LIN {X 0,Y 162.118,Z 704.88,A -85,B 0,C 180,E1 -25521.787,E2 -25521.787} C_VEL
LIN {X 0,Y 165.907,Z 693.035,A -85,B 0,C 180,E1 -25523.34,E2 -25523.34} C_VEL
LIN {X 0,Y 169.008,Z 680.232,A -85,B 0,C 180,E1 -25524.51,E2 -25524.51} C_VEL
LIN {X 0,Y 171.187,Z 667.318,A -85,B 0,C 180,E1 -25525.271,E2 -25525.271} C_VEL
LIN {X 0,Y 173.639,Z 638.606,A -85,B 0,C 180,E1 -25526.285,E2 -25526.285} C_VEL
LIN {X 0,Y 171.957,Z 634.293,A -85,B 0,C 180,E1 -25527.385,E2 -25527.385} C_VEL
LIN {X 0,Y 167.291,Z 625.497,A -85,B 0,C 180,E1 -25530.485,E2 -25530.485} C_VEL
LIN {X 0,Y 162.834,Z 618.085,A -85,B 0,C 180,E1 -25533.829,E2 -25533.829} C_VEL
LIN {X 0,Y 158.773,Z 611.768,A -85,B 0,C 180,E1 -25537.384,E2 -25537.384} C_VEL
LIN {X 0,Y 156.111,Z 607.869,A -85,B 0,C 180,E1 -25540.095,E2 -25540.095} C_VEL
LIN {X 0,Y 153.27,Z 603.781,A -85,B 0,C 180,E1 -25543.517,E2 -25543.517} C_VEL
LIN {X 0,Y 150.908,Z 600.619,A -85,B 0,C 180,E1 -25547.017,E2 -25547.017} C_VEL
LIN {X 0,Y 150.151,Z 599.126,A -85,B 0,C 180,E1 -25548.448,E2 -25548.448} C_VEL
LIN {X 0,Y 147.441,Z 595.958,A -85,B 0,C 180,E1 -25555.215,E2 -25555.215} C_VEL
LIN {X 0,Y 146.954,Z 593.781,A -85,B 0,C 180,E1 -25558.629,E2 -25558.629} C_VEL
LIN {X 0,Y 146.959,Z 593.9,A -85,B 0,C 180,E1 -25565.144,E2 -25565.144} C_VEL
LIN {X 0,Y 148.425,Z 597.823,A -85,B 0,C 180,E1 -25571.678,E2 -25571.678} C_VEL
LIN {X 0,Y 150.347,Z 599.549,A -85,B 0,C 180,E1 -25575.592,E2 -25575.592} C_VEL
LIN {X 0,Y 152.295,Z 602.878,A -85,B 0,C 180,E1 -25578.846,E2 -25578.846} C_VEL
LIN {X 0,Y 153.871,Z 604.601,A -85,B 0,C 180,E1 -25580.906,E2 -25580.906} C_VEL
LIN {X 0,Y 156.542,Z 608.421,A -85,B 0,C 180,E1 -25584.008,E2 -25584.008} C_VEL
LIN {X 0,Y 159.371,Z 612.825,A -85,B 0,C 180,E1 -25586.839,E2 -25586.839} C_VEL
LIN {X 0,Y 163.358,Z 620.37,A -85,B 0,C 180,E1 -25590.365,E2 -25590.365} C_VEL
LIN {X 0,Y 168.135,Z 630.963,A -85,B 0,C 180,E1 -25594.059,E2 -25594.059} C_VEL
LIN {X 0,Y 172.255,Z 641.448,A -85,B 0,C 180,E1 -25596.915,E2 -25596.915} C_VEL
LIN {X 0,Y 173.197,Z 644.283,A -85,B 0,C 180,E1 -25597.553,E2 -25597.553} C_VEL
LIN {X 0,Y 170.754,Z 672.948,A -85,B 0,C 180,E1 -25598.556,E2 -25598.556} C_VEL
LIN {X 0,Y 168.387,Z 686.79,A -85,B 0,C 180,E1 -25599.366,E2 -25599.366} C_VEL
LIN {X 0,Y 165.189,Z 699.4,A -85,B 0,C 180,E1 -25600.494,E2 -25600.494} C_VEL
LIN {X 0,Y 160.856,Z 711.897,A -85,B 0,C 180,E1 -25602.035,E2 -25602.035} C_VEL
LIN {X 0,Y 156.12,Z 723.049,A -85,B 0,C 180,E1 -25603.925,E2 -25603.925} C_VEL
LIN {X 0,Y 151.618,Z 732.079,A -85,B 0,C 180,E1 -25605.95,E2 -25605.95} C_VEL
LIN {X 0,Y 146.276,Z 741.359,A -85,B 0,C 180,E1 -25608.653,E2 -25608.653} C_VEL
LIN {X 0,Y 140.348,Z 750.363,A -85,B 0,C 180,E1 -25612.164,E2 -25612.164} C_VEL
LIN {X 0,Y 135.119,Z 757.631,A -85,B 0,C 180,E1 -25616.005,E2 -25616.005} C_VEL
LIN {X 0,Y 129.943,Z 764.292,A -85,B 0,C 180,E1 -25620.872,E2 -25620.872} C_VEL
LIN {X 0,Y 126.155,Z 768.706,A -85,B 0,C 180,E1 -25625.304,E2 -25625.304} C_VEL
LIN {X 0,Y 123.114,Z 772.057,A -85,B 0,C 180,E1 -25629.971,E2 -25629.971} C_VEL
LIN {X 0,Y 120.562,Z 775.013,A -85,B 0,C 180,E1 -25636.516,E2 -25636.516} C_VEL
LIN {X 0,Y 119.8,Z 775.898,A -85,B 0,C 180,E1 -25639.864,E2 -25639.864} C_VEL
LIN {X 0,Y 119.372,Z 776.351,A -85,B 0,C 180,E1 -25643.238,E2 -25643.238} C_VEL
LIN {X 0,Y 119.224,Z 776.413,A -85,B 0,C 180,E1 -25646.621,E2 -25646.621} C_VEL
LIN {X 0,Y 119.36,Z 776.091,A -85,B 0,C 180,E1 -25650,E2 -25650} C_VEL
LIN {X 0,Y 119.284,Z 775.366,A -85,B 0,C 180,E1 -25653.378,E2 -25653.378} C_VEL
LIN {X 0,Y 119.406,Z 774.199,A -85,B 0,C 180,E1 -25656.76,E2 -25656.76} C_VEL
LIN {X 0,Y 120.072,Z 771.674,A -85,B 0,C 180,E1 -25661.821,E2 -25661.821} C_VEL
LIN {X 0,Y 121.494,Z 768.132,A -85,B 0,C 180,E1 -25666.812,E2 -25666.812} C_VEL
LIN {X 0,Y 123.837,Z 763.485,A -85,B 0,C 180,E1 -25671.647,E2 -25671.647} C_VEL
LIN {X 0,Y 127.337,Z 756.895,A -85,B 0,C 180,E1 -25676.744,E2 -25676.744} C_VEL
LIN {X 0,Y 128.513,Z 753.671,A -85,B 0,C 180,E1 -25678.89,E2 -25678.89} C_VEL
LIN {X 0,Y 128.84,Z 748.046,A -85,B 0,C 180,E1 -25682.527,E2 -25682.527} C_VEL
LIN {X 0,Y 129.411,Z 741.896,A -85,B 0,C 180,E1 -25685.979,E2 -25685.979} C_VEL
LIN {X 0,Y 130.899,Z 737.763,A -85,B 0,C 180,E1 -25687.745,E2 -25687.745} C_VEL
LIN {X 0,Y 135.517,Z 727.836,A -85,B 0,C 180,E1 -25690.899,E2 -25690.899} C_VEL
LIN {X 0,Y 140.137,Z 716.363,A -85,B 0,C 180,E1 -25693.595,E2 -25693.595} C_VEL
LIN {X 0,Y 143.954,Z 705.097,A -85,B 0,C 180,E1 -25695.561,E2 -25695.561} C_VEL
LIN {X 0,Y 147.364,Z 692.405,A -85,B 0,C 180,E1 -25697.159,E2 -25697.159} C_VEL
LIN {X 0,Y 149.806,Z 679.678,A -85,B 0,C 180,E1 -25698.263,E2 -25698.263} C_VEL
LIN {X 0,Y 151.379,Z 666.349,A -85,B 0,C 180,E1 -25698.991,E2 -25698.991} C_VEL
LIN {X 0,Y 153.858,Z 633.14,A -85,B 0,C 180,E1 -25700.246,E2 -25700.246} C_VEL
LIN {X 0,Y 150.172,Z 622.407,A -85,B 0,C 180,E1 -25702.622,E2 -25702.622} C_VEL
LIN {X 0,Y 145.722,Z 611.956,A -85,B 0,C 180,E1 -25705.632,E2 -25705.632} C_VEL
LIN {X 0,Y 142.708,Z 605.888,A -85,B 0,C 180,E1 -25707.827,E2 -25707.827} C_VEL
LIN {X 0,Y 138.817,Z 599.957,A -85,B 0,C 180,E1 -25710.828,E2 -25710.828} C_VEL
LIN {X 0,Y 136.129,Z 596.114,A -85,B 0,C 180,E1 -25713.145,E2 -25713.145} C_VEL
LIN {X 0,Y 133.127,Z 591.974,A -85,B 0,C 180,E1 -25716.057,E2 -25716.057} C_VEL
LIN {X 0,Y 130.457,Z 588.575,A -85,B 0,C 180,E1 -25719.022,E2 -25719.022} C_VEL
LIN {X 0,Y 129.642,Z 587.229,A -85,B 0,C 180,E1 -25720.072,E2 -25720.072} C_VEL
LIN {X 0,Y 127.258,Z 584.922,A -85,B 0,C 180,E1 -25723.275,E2 -25723.275} C_VEL
LIN {X 0,Y 125.817,Z 582.049,A -85,B 0,C 180,E1 -25725.855,E2 -25725.855} C_VEL
LIN {X 0,Y 122.518,Z 579.199,A -85,B 0,C 180,E1 -25733.413,E2 -25733.413} C_VEL
LIN {X 0,Y 121.752,Z 576.723,A -85,B 0,C 180,E1 -25737.726,E2 -25737.726} C_VEL
LIN {X 0,Y 121.716,Z 576.23,A -85,B 0,C 180,E1 -25738.346,E2 -25738.346} C_VEL
LIN {X 0,Y 121.562,Z 576.369,A -85,B 0,C 180,E1 -25744.975,E2 -25744.975} C_VEL
LIN {X 0,Y 123.992,Z 581.142,A -85,B 0,C 180,E1 -25755.198,E2 -25755.198} C_VEL
LIN {X 0,Y 125.934,Z 582.245,A -85,B 0,C 180,E1 -25758.822,E2 -25758.822} C_VEL
LIN {X 0,Y 127.529,Z 585.423,A -85,B 0,C 180,E1 -25761.618,E2 -25761.618} C_VEL
LIN {X 0,Y 130.086,Z 587.796,A -85,B 0,C 180,E1 -25764.94,E2 -25764.94} C_VEL
LIN {X 0,Y 132.291,Z 591.204,A -85,B 0,C 180,E1 -25767.556,E2 -25767.556} C_VEL
LIN {X 0,Y 133.801,Z 592.774,A -85,B 0,C 180,E1 -25769.076,E2 -25769.076} C_VEL
LIN {X 0,Y 136.478,Z 596.545,A -85,B 0,C 180,E1 -25771.621,E2 -25771.621} C_VEL
LIN {X 0,Y 140.346,Z 602.297,A -85,B 0,C 180,E1 -25774.859,E2 -25774.859} C_VEL
LIN {X 0,Y 144.7,Z 609.144,A -85,B 0,C 180,E1 -25778.042,E2 -25778.042} C_VEL
LIN {X 0,Y 149.212,Z 617.122,A -85,B 0,C 180,E1 -25780.99,E2 -25780.99} C_VEL
LIN {X 0,Y 153.985,Z 626.915,A -85,B 0,C 180,E1 -25783.837,E2 -25783.837} C_VEL
LIN {X 0,Y 154.23,Z 628.253,A -85,B 0,C 180,E1 -25784.032,E2 -25784.032} C_VEL
LIN {X 0,Y 151.162,Z 666.895,A -85,B 0,C 180,E1 -25785.536,E2 -25785.536} C_VEL
LIN {X 0,Y 149.109,Z 680.278,A -85,B 0,C 180,E1 -25786.482,E2 -25786.482} C_VEL
LIN {X 0,Y 146.492,Z 692.384,A -85,B 0,C 180,E1 -25787.807,E2 -25787.807} C_VEL
LIN {X 0,Y 143.233,Z 703.52,A -85,B 0,C 180,E1 -25789.449,E2 -25789.449} C_VEL
LIN {X 0,Y 139.286,Z 715.044,A -85,B 0,C 180,E1 -25791.823,E2 -25791.823} C_VEL
LIN {X 0,Y 134.978,Z 725.424,A -85,B 0,C 180,E1 -25794.603,E2 -25794.603} C_VEL
LIN {X 0,Y 130.826,Z 733.925,A -85,B 0,C 180,E1 -25797.507,E2 -25797.507} C_VEL
LIN {X 0,Y 126.685,Z 741.757,A -85,B 0,C 180,E1 -25800.961,E2 -25800.961} C_VEL
LIN {X 0,Y 122.587,Z 749.395,A -85,B 0,C 180,E1 -25805.441,E2 -25805.441} C_VEL
LIN {X 0,Y 118.556,Z 756.43,A -85,B 0,C 180,E1 -25810.972,E2 -25810.972} C_VEL
LIN {X 0,Y 115.874,Z 761.117,A -85,B 0,C 180,E1 -25815.96,E2 -25815.96} C_VEL
LIN {X 0,Y 113.867,Z 764.711,A -85,B 0,C 180,E1 -25821.124,E2 -25821.124} C_VEL
LIN {X 0,Y 112.581,Z 767.627,A -85,B 0,C 180,E1 -25827.226,E2 -25827.226} C_VEL
LIN {X 0,Y 112.176,Z 769.339,A -85,B 0,C 180,E1 -25833.592,E2 -25833.592} C_VEL
LIN {X 0,Y 112.24,Z 769.739,A -85,B 0,C 180,E1 -25837.194,E2 -25837.194} C_VEL
LIN {X 0,Y 112.619,Z 769.76,A -85,B 0,C 180,E1 -25840.79,E2 -25840.79} C_VEL
LIN {X 0,Y 113.276,Z 769.401,A -85,B 0,C 180,E1 -25844.369,E2 -25844.369} C_VEL
LIN {X 0,Y 114.271,Z 768.638,A -85,B 0,C 180,E1 -25847.909,E2 -25847.909} C_VEL
LIN {X 0,Y 117.478,Z 765.84,A -85,B 0,C 180,E1 -25854.756,E2 -25854.756} C_VEL
LIN {X 0,Y 120.696,Z 762.736,A -85,B 0,C 180,E1 -25859.474,E2 -25859.474} C_VEL
LIN {X 0,Y 124.879,Z 758.31,A -85,B 0,C 180,E1 -25864.248,E2 -25864.248} C_VEL
LIN {X 0,Y 129.683,Z 752.804,A -85,B 0,C 180,E1 -25868.551,E2 -25868.551} C_VEL
LIN {X 0,Y 135.205,Z 745.915,A -85,B 0,C 180,E1 -25872.511,E2 -25872.511} C_VEL
LIN {X 0,Y 140.125,Z 738.86,A -85,B 0,C 180,E1 -25875.618,E2 -25875.618} C_VEL
LIN {X 0,Y 145.46,Z 730.317,A -85,B 0,C 180,E1 -25878.493,E2 -25878.493} C_VEL
LIN {X 0,Y 150.579,Z 720.926,A -85,B 0,C 180,E1 -25880.889,E2 -25880.889} C_VEL
LIN {X 0,Y 155.981,Z 709.252,A -85,B 0,C 180,E1 -25883.105,E2 -25883.105} C_VEL
LIN {X 0,Y 160.204,Z 697.641,A -85,B 0,C 180,E1 -25884.79,E2 -25884.79} C_VEL
LIN {X 0,Y 163.634,Z 685.457,A -85,B 0,C 180,E1 -25886.058,E2 -25886.058} C_VEL
LIN {X 0,Y 166.304,Z 672.324,A -85,B 0,C 180,E1 -25886.991,E2 -25886.991} C_VEL
LIN {X 0,Y 167.9,Z 659.529,A -85,B 0,C 180,E1 -25887.531,E2 -25887.531} C_VEL
LIN {X 0,Y 169.328,Z 640.85,A -85,B 0,C 180,E1 -25888.206,E2 -25888.206} C_VEL
LIN {X 0,Y 165.427,Z 632.926,A -85,B 0,C 180,E1 -25890.938,E2 -25890.938} C_VEL
LIN {X 0,Y 161.192,Z 625.29,A -85,B 0,C 180,E1 -25894.259,E2 -25894.259} C_VEL
LIN {X 0,Y 157.108,Z 618.499,A -85,B 0,C 180,E1 -25897.997,E2 -25897.997} C_VEL
LIN {X 0,Y 154.077,Z 614.001,A -85,B 0,C 180,E1 -25901.262,E2 -25901.262} C_VEL
LIN {X 0,Y 151.71,Z 610.394,A -85,B 0,C 180,E1 -25904.337,E2 -25904.337} C_VEL
LIN {X 0,Y 149.37,Z 606.945,A -85,B 0,C 180,E1 -25908.12,E2 -25908.12} C_VEL
LIN {X 0,Y 148.887,Z 605.947,A -85,B 0,C 180,E1 -25909.116,E2 -25909.116} C_VEL
LIN {X 0,Y 146.412,Z 602.783,A -85,B 0,C 180,E1 -25915.871,E2 -25915.871} C_VEL
LIN {X 0,Y 146.008,Z 600.763,A -85,B 0,C 180,E1 -25919.31,E2 -25919.31} C_VEL
LIN {X 0,Y 146.037,Z 601.034,A -85,B 0,C 180,E1 -25924.831,E2 -25924.831} C_VEL
LIN {X 0,Y 147.563,Z 604.989,A -85,B 0,C 180,E1 -25931.747,E2 -25931.747} C_VEL
LIN {X 0,Y 149.034,Z 606.321,A -85,B 0,C 180,E1 -25934.857,E2 -25934.857} C_VEL
LIN {X 0,Y 151.098,Z 609.827,A -85,B 0,C 180,E1 -25938.467,E2 -25938.467} C_VEL
LIN {X 0,Y 152.264,Z 611.208,A -85,B 0,C 180,E1 -25940.077,E2 -25940.077} C_VEL
LIN {X 0,Y 155.367,Z 615.93,A -85,B 0,C 180,E1 -25943.846,E2 -25943.846} C_VEL
LIN {X 0,Y 157.331,Z 619.197,A -85,B 0,C 180,E1 -25945.908,E2 -25945.908} C_VEL
LIN {X 0,Y 160.981,Z 626.578,A -85,B 0,C 180,E1 -25949.365,E2 -25949.365} C_VEL
LIN {X 0,Y 165.062,Z 636.16,A -85,B 0,C 180,E1 -25952.764,E2 -25952.764} C_VEL
LIN {X 0,Y 168.692,Z 645.914,A -85,B 0,C 180,E1 -25955.497,E2 -25955.497} C_VEL
LIN {X 0,Y 168.933,Z 646.687,A -85,B 0,C 180,E1 -25955.676,E2 -25955.676} C_VEL
LIN {X 0,Y 166.573,Z 673.039,A -85,B 0,C 180,E1 -25956.609,E2 -25956.609} C_VEL
LIN {X 0,Y 164.128,Z 686.751,A -85,B 0,C 180,E1 -25957.406,E2 -25957.406} C_VEL
LIN {X 0,Y 161.016,Z 698.742,A -85,B 0,C 180,E1 -25958.472,E2 -25958.472} C_VEL
LIN {X 0,Y 156.829,Z 710.545,A -85,B 0,C 180,E1 -25959.878,E2 -25959.878} C_VEL
LIN {X 0,Y 152.527,Z 720.615,A -85,B 0,C 180,E1 -25961.519,E2 -25961.519} C_VEL
LIN {X 0,Y 147.209,Z 731.097,A -85,B 0,C 180,E1 -25963.774,E2 -25963.774} C_VEL
LIN {X 0,Y 142.094,Z 739.672,A -85,B 0,C 180,E1 -25966.178,E2 -25966.178} C_VEL
LIN {X 0,Y 136.811,Z 747.585,A -85,B 0,C 180,E1 -25969.084,E2 -25969.084} C_VEL
LIN {X 0,Y 131.026,Z 755.339,A -85,B 0,C 180,E1 -25972.885,E2 -25972.885} C_VEL
LIN {X 0,Y 125.275,Z 762.475,A -85,B 0,C 180,E1 -25977.796,E2 -25977.796} C_VEL
LIN {X 0,Y 120.945,Z 767.245,A -85,B 0,C 180,E1 -25982.299,E2 -25982.299} C_VEL
LIN {X 0,Y 117.455,Z 770.911,A -85,B 0,C 180,E1 -25987.113,E2 -25987.113} C_VEL
LIN {X 0,Y 114.859,Z 773.578,A -85,B 0,C 180,E1 -25992.186,E2 -25992.186} C_VEL
LIN {X 0,Y 113.653,Z 774.846,A -85,B 0,C 180,E1 -25995.68,E2 -25995.68} C_VEL
LIN {X 0,Y 112.791,Z 775.714,A -85,B 0,C 180,E1 -25999.227,E2 -25999.227} C_VEL
LIN {X 0,Y 112.3,Z 776.151,A -85,B 0,C 180,E1 -26002.81,E2 -26002.81} C_VEL
LIN {X 0,Y 112.132,Z 776.202,A -85,B 0,C 180,E1 -26006.407,E2 -26006.407} C_VEL
LIN {X 0,Y 112.261,Z 775.87,A -85,B 0,C 180,E1 -26010,E2 -26010} C_VEL
LIN {X 0,Y 112.181,Z 775.131,A -85,B 0,C 180,E1 -26013.592,E2 -26013.592} C_VEL
LIN {X 0,Y 112.325,Z 773.944,A -85,B 0,C 180,E1 -26017.188,E2 -26017.188} C_VEL
LIN {X 0,Y 113.119,Z 771.397,A -85,B 0,C 180,E1 -26022.559,E2 -26022.559} C_VEL
LIN {X 0,Y 114.666,Z 767.829,A -85,B 0,C 180,E1 -26027.845,E2 -26027.845} C_VEL
LIN {X 0,Y 117.227,Z 763.156,A -85,B 0,C 180,E1 -26032.934,E2 -26032.934} C_VEL
LIN {X 0,Y 121.3,Z 756.107,A -85,B 0,C 180,E1 -26038.554,E2 -26038.554} C_VEL
LIN {X 0,Y 125.585,Z 748.276,A -85,B 0,C 180,E1 -26043.195,E2 -26043.195} C_VEL
LIN {X 0,Y 130.351,Z 738.851,A -85,B 0,C 180,E1 -26047.34,E2 -26047.34} C_VEL
LIN {X 0,Y 130.899,Z 737.763,A -85,B 0,C 180,E1 -26047.745,E2 -26047.745} C_VEL
LIN {X 0,Y 132.468,Z 733.502,A -85,B 0,C 180,E1 -26049.393,E2 -26049.393} C_VEL
LIN {X 0,Y 133.545,Z 726.254,A -85,B 0,C 180,E1 -26052.276,E2 -26052.276} C_VEL
LIN {X 0,Y 134.543,Z 718.538,A -85,B 0,C 180,E1 -26054.911,E2 -26054.911} C_VEL
LIN {X 0,Y 135.908,Z 713.543,A -85,B 0,C 180,E1 -26056.123,E2 -26056.123} C_VEL
LIN {X 0,Y 139.62,Z 702.498,A -85,B 0,C 180,E1 -26057.94,E2 -26057.94} C_VEL
LIN {X 0,Y 142.901,Z 690.176,A -85,B 0,C 180,E1 -26059.395,E2 -26059.395} C_VEL
LIN {X 0,Y 145.439,Z 676.771,A -85,B 0,C 180,E1 -26060.475,E2 -26060.475} C_VEL
LIN {X 0,Y 147.034,Z 661.516,A -85,B 0,C 180,E1 -26061.184,E2 -26061.184} C_VEL
LIN {X 0,Y 149.056,Z 635.163,A -85,B 0,C 180,E1 -26062.197,E2 -26062.197} C_VEL
LIN {X 0,Y 145.717,Z 625.389,A -85,B 0,C 180,E1 -26064.558,E2 -26064.558} C_VEL
LIN {X 0,Y 141.696,Z 615.626,A -85,B 0,C 180,E1 -26067.569,E2 -26067.569} C_VEL
LIN {X 0,Y 139.318,Z 610.734,A -85,B 0,C 180,E1 -26069.469,E2 -26069.469} C_VEL
LIN {X 0,Y 135.869,Z 605.405,A -85,B 0,C 180,E1 -26072.36,E2 -26072.36} C_VEL
LIN {X 0,Y 133.665,Z 602.102,A -85,B 0,C 180,E1 -26074.423,E2 -26074.423} C_VEL
LIN {X 0,Y 130.973,Z 598.258,A -85,B 0,C 180,E1 -26077.236,E2 -26077.236} C_VEL
LIN {X 0,Y 128.33,Z 594.498,A -85,B 0,C 180,E1 -26080.459,E2 -26080.459} C_VEL
LIN {X 0,Y 127.249,Z 593.323,A -85,B 0,C 180,E1 -26081.901,E2 -26081.901} C_VEL
LIN {X 0,Y 125.12,Z 590.482,A -85,B 0,C 180,E1 -26085.268,E2 -26085.268} C_VEL
LIN {X 0,Y 124.286,Z 588.847,A -85,B 0,C 180,E1 -26086.928,E2 -26086.928} C_VEL
LIN {X 0,Y 121.121,Z 585.317,A -85,B 0,C 180,E1 -26095.633,E2 -26095.633} C_VEL
LIN {X 0,Y 120.763,Z 583.221,A -85,B 0,C 180,E1 -26099.063,E2 -26099.063} C_VEL
LIN {X 0,Y 120.66,Z 583.415,A -85,B 0,C 180,E1 -26104.594,E2 -26104.594} C_VEL
LIN {X 0,Y 122.966,Z 588.141,A -85,B 0,C 180,E1 -26114.904,E2 -26114.904} C_VEL
LIN {X 0,Y 124.511,Z 589.209,A -85,B 0,C 180,E1 -26117.98,E2 -26117.98} C_VEL
LIN {X 0,Y 126.347,Z 592.521,A -85,B 0,C 180,E1 -26121.282,E2 -26121.282} C_VEL
LIN {X 0,Y 128.309,Z 594.45,A -85,B 0,C 180,E1 -26123.967,E2 -26123.967} C_VEL
LIN {X 0,Y 130.779,Z 598.091,A -85,B 0,C 180,E1 -26127.016,E2 -26127.016} C_VEL
LIN {X 0,Y 131.935,Z 599.597,A -85,B 0,C 180,E1 -26128.268,E2 -26128.268} C_VEL
LIN {X 0,Y 135.326,Z 604.562,A -85,B 0,C 180,E1 -26131.605,E2 -26131.605} C_VEL
LIN {X 0,Y 139.788,Z 611.578,A -85,B 0,C 180,E1 -26135.366,E2 -26135.366} C_VEL
LIN {X 0,Y 144.244,Z 619.402,A -85,B 0,C 180,E1 -26138.642,E2 -26138.642} C_VEL
LIN {X 0,Y 148.524,Z 628.114,A -85,B 0,C 180,E1 -26141.489,E2 -26141.489} C_VEL
LIN {X 0,Y 149.367,Z 629.964,A -85,B 0,C 180,E1 -26142.021,E2 -26142.021} C_VEL
LIN {X 0,Y 146.401,Z 666.845,A -85,B 0,C 180,E1 -26143.502,E2 -26143.502} C_VEL
LIN {X 0,Y 144.324,Z 680.033,A -85,B 0,C 180,E1 -26144.43,E2 -26144.43} C_VEL
LIN {X 0,Y 141.609,Z 692.171,A -85,B 0,C 180,E1 -26145.749,E2 -26145.749} C_VEL
LIN {X 0,Y 137.946,Z 704.19,A -85,B 0,C 180,E1 -26147.543,E2 -26147.543} C_VEL
LIN {X 0,Y 133.81,Z 715.628,A -85,B 0,C 180,E1 -26149.956,E2 -26149.956} C_VEL
LIN {X 0,Y 129.271,Z 725.945,A -85,B 0,C 180,E1 -26152.785,E2 -26152.785} C_VEL
LIN {X 0,Y 124.925,Z 734.392,A -85,B 0,C 180,E1 -26155.767,E2 -26155.767} C_VEL
LIN {X 0,Y 120.559,Z 742.177,A -85,B 0,C 180,E1 -26159.331,E2 -26159.331} C_VEL
LIN {X 0,Y 116.199,Z 749.764,A -85,B 0,C 180,E1 -26163.993,E2 -26163.993} C_VEL
LIN {X 0,Y 111.886,Z 756.768,A -85,B 0,C 180,E1 -26169.79,E2 -26169.79} C_VEL
LIN {X 0,Y 109.024,Z 761.427,A -85,B 0,C 180,E1 -26175.058,E2 -26175.058} C_VEL
LIN {X 0,Y 106.875,Z 764.995,A -85,B 0,C 180,E1 -26180.538,E2 -26180.538} C_VEL
LIN {X 0,Y 105.625,Z 767.56,A -85,B 0,C 180,E1 -26186.185,E2 -26186.185} C_VEL
LIN {X 0,Y 105.222,Z 768.772,A -85,B 0,C 180,E1 -26190,E2 -26190} C_VEL
LIN {X 0,Y 105.09,Z 769.561,A -85,B 0,C 180,E1 -26193.834,E2 -26193.834} C_VEL
LIN {X 0,Y 105.607,Z 769.96,A -85,B 0,C 180,E1 -26201.516,E2 -26201.516} C_VEL
LIN {X 0,Y 106.366,Z 769.589,A -85,B 0,C 180,E1 -26205.325,E2 -26205.325} C_VEL
LIN {X 0,Y 107.48,Z 768.803,A -85,B 0,C 180,E1 -26209.083,E2 -26209.083} C_VEL
LIN {X 0,Y 111.021,Z 765.979,A -85,B 0,C 180,E1 -26216.303,E2 -26216.303} C_VEL
LIN {X 0,Y 114.641,Z 762.727,A -85,B 0,C 180,E1 -26221.404,E2 -26221.404} C_VEL
LIN {X 0,Y 119.028,Z 758.396,A -85,B 0,C 180,E1 -26226.188,E2 -26226.188} C_VEL
LIN {X 0,Y 124.187,Z 752.86,A -85,B 0,C 180,E1 -26230.602,E2 -26230.602} C_VEL
LIN {X 0,Y 130.021,Z 745.932,A -85,B 0,C 180,E1 -26234.642,E2 -26234.642} C_VEL
LIN {X 0,Y 135.216,Z 738.839,A -85,B 0,C 180,E1 -26237.786,E2 -26237.786} C_VEL
LIN {X 0,Y 140.822,Z 730.233,A -85,B 0,C 180,E1 -26240.673,E2 -26240.673} C_VEL
LIN {X 0,Y 146.19,Z 720.782,A -85,B 0,C 180,E1 -26243.056,E2 -26243.056} C_VEL
LIN {X 0,Y 151.803,Z 709.033,A -85,B 0,C 180,E1 -26245.26,E2 -26245.26} C_VEL
LIN {X 0,Y 156.202,Z 697.255,A -85,B 0,C 180,E1 -26246.927,E2 -26246.927} C_VEL
LIN {X 0,Y 160.011,Z 683.903,A -85,B 0,C 180,E1 -26248.261,E2 -26248.261} C_VEL
LIN {X 0,Y 162.54,Z 671.326,A -85,B 0,C 180,E1 -26249.105,E2 -26249.105} C_VEL
LIN {X 0,Y 164.297,Z 656.044,A -85,B 0,C 180,E1 -26249.693,E2 -26249.693} C_VEL
LIN {X 0,Y 165.281,Z 644.004,A -85,B 0,C 180,E1 -26250.116,E2 -26250.116} C_VEL
LIN {X 0,Y 161.383,Z 636.036,A -85,B 0,C 180,E1 -26253.139,E2 -26253.139} C_VEL
LIN {X 0,Y 157.306,Z 628.511,A -85,B 0,C 180,E1 -26256.758,E2 -26256.758} C_VEL
LIN {X 0,Y 154.155,Z 623.384,A -85,B 0,C 180,E1 -26260.005,E2 -26260.005} C_VEL
LIN {X 0,Y 152.317,Z 620.42,A -85,B 0,C 180,E1 -26262.2,E2 -26262.2} C_VEL
LIN {X 0,Y 150.209,Z 617.008,A -85,B 0,C 180,E1 -26265.139,E2 -26265.139} C_VEL
LIN {X 0,Y 147.978,Z 613.477,A -85,B 0,C 180,E1 -26269.048,E2 -26269.048} C_VEL
LIN {X 0,Y 147.655,Z 612.811,A -85,B 0,C 180,E1 -26269.764,E2 -26269.764} C_VEL
LIN {X 0,Y 145.347,Z 609.414,A -85,B 0,C 180,E1 -26276.881,E2 -26276.881} C_VEL
LIN {X 0,Y 145.084,Z 607.736,A -85,B 0,C 180,E1 -26280,E2 -26280} C_VEL
LIN {X 0,Y 145.126,Z 608.106,A -85,B 0,C 180,E1 -26284.513,E2 -26284.513} C_VEL
LIN {X 0,Y 146.558,Z 611.977,A -85,B 0,C 180,E1 -26291.443,E2 -26291.443} C_VEL
LIN {X 0,Y 147.821,Z 613.259,A -85,B 0,C 180,E1 -26294.278,E2 -26294.278} C_VEL
LIN {X 0,Y 150.016,Z 616.928,A -85,B 0,C 180,E1 -26298.246,E2 -26298.246} C_VEL
LIN {X 0,Y 150.811,Z 618.052,A -85,B 0,C 180,E1 -26299.414,E2 -26299.414} C_VEL
LIN {X 0,Y 153.565,Z 622.404,A -85,B 0,C 180,E1 -26302.961,E2 -26302.961} C_VEL
LIN {X 0,Y 155.319,Z 625.553,A -85,B 0,C 180,E1 -26304.938,E2 -26304.938} C_VEL
LIN {X 0,Y 158.636,Z 632.734,A -85,B 0,C 180,E1 -26308.316,E2 -26308.316} C_VEL
LIN {X 0,Y 162.266,Z 641.896,A -85,B 0,C 180,E1 -26311.584,E2 -26311.584} C_VEL
LIN {X 0,Y 164.853,Z 649.208,A -85,B 0,C 180,E1 -26313.711,E2 -26313.711} C_VEL
LIN {X 0,Y 162.636,Z 672.86,A -85,B 0,C 180,E1 -26314.552,E2 -26314.552} C_VEL
LIN {X 0,Y 160.16,Z 686.381,A -85,B 0,C 180,E1 -26315.331,E2 -26315.331} C_VEL
LIN {X 0,Y 156.708,Z 699.085,A -85,B 0,C 180,E1 -26316.444,E2 -26316.444} C_VEL
LIN {X 0,Y 152.391,Z 710.773,A -85,B 0,C 180,E1 -26317.837,E2 -26317.837} C_VEL
LIN {X 0,Y 147.915,Z 720.765,A -85,B 0,C 180,E1 -26319.459,E2 -26319.459} C_VEL
LIN {X 0,Y 142.398,Z 731.185,A -85,B 0,C 180,E1 -26321.714,E2 -26321.714} C_VEL
LIN {X 0,Y 137.062,Z 739.711,A -85,B 0,C 180,E1 -26324.123,E2 -26324.123} C_VEL
LIN {X 0,Y 131.536,Z 747.584,A -85,B 0,C 180,E1 -26327.061,E2 -26327.061} C_VEL
LIN {X 0,Y 125.418,Z 755.287,A -85,B 0,C 180,E1 -26330.92,E2 -26330.92} C_VEL
LIN {X 0,Y 120.084,Z 761.494,A -85,B 0,C 180,E1 -26335.218,E2 -26335.218} C_VEL
LIN {X 0,Y 114.679,Z 767.136,A -85,B 0,C 180,E1 -26340.642,E2 -26340.642} C_VEL
LIN {X 0,Y 110.936,Z 770.778,A -85,B 0,C 180,E1 -26345.683,E2 -26345.683} C_VEL
LIN {X 0,Y 108.077,Z 773.421,A -85,B 0,C 180,E1 -26351.027,E2 -26351.027} C_VEL
LIN {X 0,Y 106.761,Z 774.679,A -85,B 0,C 180,E1 -26354.733,E2 -26354.733} C_VEL
LIN {X 0,Y 105.812,Z 775.528,A -85,B 0,C 180,E1 -26358.507,E2 -26358.507} C_VEL
LIN {X 0,Y 105.252,Z 775.952,A -85,B 0,C 180,E1 -26362.326,E2 -26362.326} C_VEL
LIN {X 0,Y 105.04,Z 775.992,A -85,B 0,C 180,E1 -26366.164,E2 -26366.164} C_VEL
LIN {X 0,Y 105.173,Z 775.649,A -85,B 0,C 180,E1 -26370,E2 -26370} C_VEL
LIN {X 0,Y 105.097,Z 774.893,A -85,B 0,C 180,E1 -26373.834,E2 -26373.834} C_VEL
LIN {X 0,Y 105.267,Z 773.689,A -85,B 0,C 180,E1 -26377.673,E2 -26377.673} C_VEL
LIN {X 0,Y 106.157,Z 771.118,A -85,B 0,C 180,E1 -26383.398,E2 -26383.398} C_VEL
LIN {X 0,Y 107.884,Z 767.526,A -85,B 0,C 180,E1 -26389.009,E2 -26389.009} C_VEL
LIN {X 0,Y 110.692,Z 762.827,A -85,B 0,C 180,E1 -26394.374,E2 -26394.374} C_VEL
LIN {X 0,Y 114.369,Z 756.873,A -85,B 0,C 180,E1 -26399.445,E2 -26399.445} C_VEL
LIN {X 0,Y 118.746,Z 749.443,A -85,B 0,C 180,E1 -26404.209,E2 -26404.209} C_VEL
LIN {X 0,Y 123.816,Z 740.194,A -85,B 0,C 180,E1 -26408.636,E2 -26408.636} C_VEL
LIN {X 0,Y 129.181,Z 729.51,A -85,B 0,C 180,E1 -26412.317,E2 -26412.317} C_VEL
LIN {X 0,Y 133.951,Z 718.618,A -85,B 0,C 180,E1 -26415.096,E2 -26415.096} C_VEL
LIN {X 0,Y 135.908,Z 713.543,A -85,B 0,C 180,E1 -26416.123,E2 -26416.123} C_VEL
LIN {X 0,Y 137.179,Z 708.426,A -85,B 0,C 180,E1 -26417.262,E2 -26417.262} C_VEL
LIN {X 0,Y 137.771,Z 699.917,A -85,B 0,C 180,E1 -26419.439,E2 -26419.439} C_VEL
LIN {X 0,Y 138.237,Z 691.126,A -85,B 0,C 180,E1 -26421.318,E2 -26421.318} C_VEL
LIN {X 0,Y 139.21,Z 685.539,A -85,B 0,C 180,E1 -26421.962,E2 -26421.962} C_VEL
LIN {X 0,Y 141.398,Z 672.552,A -85,B 0,C 180,E1 -26422.862,E2 -26422.862} C_VEL
LIN {X 0,Y 144.429,Z 637.273,A -85,B 0,C 180,E1 -26424.273,E2 -26424.273} C_VEL
LIN {X 0,Y 141.408,Z 628.202,A -85,B 0,C 180,E1 -26426.646,E2 -26426.646} C_VEL
LIN {X 0,Y 137.488,Z 618.394,A -85,B 0,C 180,E1 -26429.934,E2 -26429.934} C_VEL
LIN {X 0,Y 134.313,Z 612.689,A -85,B 0,C 180,E1 -26432.753,E2 -26432.753} C_VEL
LIN {X 0,Y 130.882,Z 607.553,A -85,B 0,C 180,E1 -26436.159,E2 -26436.159} C_VEL
LIN {X 0,Y 128.932,Z 604.537,A -85,B 0,C 180,E1 -26438.399,E2 -26438.399} C_VEL
LIN {X 0,Y 126.105,Z 600.363,A -85,B 0,C 180,E1 -26442.177,E2 -26442.177} C_VEL
LIN {X 0,Y 123.74,Z 597.337,A -85,B 0,C 180,E1 -26446.045,E2 -26446.045} C_VEL
LIN {X 0,Y 122.977,Z 595.681,A -85,B 0,C 180,E1 -26447.695,E2 -26447.695} C_VEL
LIN {X 0,Y 120.102,Z 592.13,A -85,B 0,C 180,E1 -26456.41,E2 -26456.41} C_VEL
LIN {X 0,Y 119.813,Z 590.196,A -85,B 0,C 180,E1 -26460,E2 -26460} C_VEL
LIN {X 0,Y 119.757,Z 590.455,A -85,B 0,C 180,E1 -26464.122,E2 -26464.122} C_VEL
LIN {X 0,Y 121.867,Z 595.081,A -85,B 0,C 180,E1 -26474.424,E2 -26474.424} C_VEL
LIN {X 0,Y 123.174,Z 596.153,A -85,B 0,C 180,E1 -26477.217,E2 -26477.217} C_VEL
LIN {X 0,Y 124.999,Z 599.373,A -85,B 0,C 180,E1 -26480.664,E2 -26480.664} C_VEL
LIN {X 0,Y 126.612,Z 601.148,A -85,B 0,C 180,E1 -26483.025,E2 -26483.025} C_VEL
LIN {X 0,Y 129.255,Z 604.953,A -85,B 0,C 180,E1 -26486.436,E2 -26486.436} C_VEL
LIN {X 0,Y 132.812,Z 610.461,A -85,B 0,C 180,E1 -26490.285,E2 -26490.285} C_VEL
LIN {X 0,Y 136.777,Z 616.923,A -85,B 0,C 180,E1 -26493.904,E2 -26493.904} C_VEL
LIN {X 0,Y 140.997,Z 624.708,A -85,B 0,C 180,E1 -26497.273,E2 -26497.273} C_VEL
LIN {X 0,Y 144.711,Z 632.63,A -85,B 0,C 180,E1 -26499.959,E2 -26499.959} C_VEL
LIN {X 0,Y 141.737,Z 667.591,A -85,B 0,C 180,E1 -26501.382,E2 -26501.382} C_VEL
LIN {X 0,Y 139.588,Z 680.578,A -85,B 0,C 180,E1 -26502.312,E2 -26502.312} C_VEL
LIN {X 0,Y 136.634,Z 693.037,A -85,B 0,C 180,E1 -26503.683,E2 -26503.683} C_VEL
LIN {X 0,Y 132.82,Z 704.86,A -85,B 0,C 180,E1 -26505.485,E2 -26505.485} C_VEL
LIN {X 0,Y 128.472,Z 716.213,A -85,B 0,C 180,E1 -26507.924,E2 -26507.924} C_VEL
LIN {X 0,Y 123.711,Z 726.464,A -85,B 0,C 180,E1 -26510.802,E2 -26510.802} C_VEL
LIN {X 0,Y 119.153,Z 734.854,A -85,B 0,C 180,E1 -26513.856,E2 -26513.856} C_VEL
LIN {X 0,Y 113.71,Z 743.938,A -85,B 0,C 180,E1 -26518.309,E2 -26518.309} C_VEL
LIN {X 0,Y 109.166,Z 751.241,A -85,B 0,C 180,E1 -26523.215,E2 -26523.215} C_VEL
LIN {X 0,Y 105.266,Z 757.106,A -85,B 0,C 180,E1 -26528.457,E2 -26528.457} C_VEL
LIN {X 0,Y 102.192,Z 761.737,A -85,B 0,C 180,E1 -26534.033,E2 -26534.033} C_VEL
LIN {X 0,Y 99.895,Z 765.278,A -85,B 0,C 180,E1 -26539.87,E2 -26539.87} C_VEL
LIN {X 0,Y 98.562,Z 767.818,A -85,B 0,C 180,E1 -26545.911,E2 -26545.911} C_VEL
LIN {X 0,Y 98.14,Z 769.016,A -85,B 0,C 180,E1 -26550,E2 -26550} C_VEL
LIN {X 0,Y 98.001,Z 769.784,A -85,B 0,C 180,E1 -26554.112,E2 -26554.112} C_VEL
LIN {X 0,Y 98.628,Z 770.159,A -85,B 0,C 180,E1 -26562.343,E2 -26562.343} C_VEL
LIN {X 0,Y 99.498,Z 769.777,A -85,B 0,C 180,E1 -26566.411,E2 -26566.411} C_VEL
LIN {X 0,Y 100.74,Z 768.967,A -85,B 0,C 180,E1 -26570.414,E2 -26570.414} C_VEL
LIN {X 0,Y 102.515,Z 767.743,A -85,B 0,C 180,E1 -26574.288,E2 -26574.288} C_VEL
LIN {X 0,Y 106.851,Z 764.327,A -85,B 0,C 180,E1 -26581.232,E2 -26581.232} C_VEL
LIN {X 0,Y 111.662,Z 760.085,A -85,B 0,C 180,E1 -26586.721,E2 -26586.721} C_VEL
LIN {X 0,Y 117.858,Z 753.923,A -85,B 0,C 180,E1 -26592.132,E2 -26592.132} C_VEL
LIN {X 0,Y 123.971,Z 747.193,A -85,B 0,C 180,E1 -26596.285,E2 -26596.285} C_VEL
LIN {X 0,Y 130.504,Z 738.811,A -85,B 0,C 180,E1 -26600.119,E2 -26600.119} C_VEL
LIN {X 0,Y 136.404,Z 730.148,A -85,B 0,C 180,E1 -26602.996,E2 -26602.996} C_VEL
LIN {X 0,Y 142.027,Z 720.639,A -85,B 0,C 180,E1 -26605.351,E2 -26605.351} C_VEL
LIN {X 0,Y 147.204,Z 710.245,A -85,B 0,C 180,E1 -26607.294,E2 -26607.294} C_VEL
LIN {X 0,Y 151.762,Z 698.821,A -85,B 0,C 180,E1 -26608.949,E2 -26608.949} C_VEL
LIN {X 0,Y 155.504,Z 686.697,A -85,B 0,C 180,E1 -26610.208,E2 -26610.208} C_VEL
LIN {X 0,Y 158.524,Z 672.973,A -85,B 0,C 180,E1 -26611.174,E2 -26611.174} C_VEL
LIN {X 0,Y 160.277,Z 660.038,A -85,B 0,C 180,E1 -26611.702,E2 -26611.702} C_VEL
LIN {X 0,Y 161.344,Z 647.14,A -85,B 0,C 180,E1 -26612.172,E2 -26612.172} C_VEL
LIN {X 0,Y 157.564,Z 639.279,A -85,B 0,C 180,E1 -26615.456,E2 -26615.456} C_VEL
LIN {X 0,Y 154.003,Z 632.691,A -85,B 0,C 180,E1 -26619.025,E2 -26619.025} C_VEL
LIN {X 0,Y 150.805,Z 627.112,A -85,B 0,C 180,E1 -26622.891,E2 -26622.891} C_VEL
LIN {X 0,Y 148.512,Z 623.365,A -85,B 0,C 180,E1 -26626.313,E2 -26626.313} C_VEL
LIN {X 0,Y 146.442,Z 619.669,A -85,B 0,C 180,E1 -26630.423,E2 -26630.423} C_VEL
LIN {X 0,Y 144.294,Z 615.857,A -85,B 0,C 180,E1 -26638.255,E2 -26638.255} C_VEL
LIN {X 0,Y 144.219,Z 614.776,A -85,B 0,C 180,E1 -26640,E2 -26640} C_VEL
LIN {X 0,Y 144.216,Z 615.073,A -85,B 0,C 180,E1 -26644.017,E2 -26644.017} C_VEL
LIN {X 0,Y 145.557,Z 618.959,A -85,B 0,C 180,E1 -26651.135,E2 -26651.135} C_VEL
LIN {X 0,Y 146.564,Z 620.024,A -85,B 0,C 180,E1 -26653.54,E2 -26653.54} C_VEL
LIN {X 0,Y 148.701,Z 623.733,A -85,B 0,C 180,E1 -26657.657,E2 -26657.657} C_VEL
LIN {X 0,Y 151.911,Z 629.021,A -85,B 0,C 180,E1 -26662.187,E2 -26662.187} C_VEL
LIN {X 0,Y 153.531,Z 632.273,A -85,B 0,C 180,E1 -26664.149,E2 -26664.149} C_VEL
LIN {X 0,Y 156.664,Z 639.637,A -85,B 0,C 180,E1 -26667.556,E2 -26667.556} C_VEL
LIN {X 0,Y 160.083,Z 649.171,A -85,B 0,C 180,E1 -26670.857,E2 -26670.857} C_VEL
LIN {X 0,Y 160.975,Z 651.803,A -85,B 0,C 180,E1 -26671.654,E2 -26671.654} C_VEL
LIN {X 0,Y 158.77,Z 673.737,A -85,B 0,C 180,E1 -26672.45,E2 -26672.45} C_VEL
LIN {X 0,Y 156.364,Z 686.126,A -85,B 0,C 180,E1 -26673.147,E2 -26673.147} C_VEL
LIN {X 0,Y 152.967,Z 698.43,A -85,B 0,C 180,E1 -26674.21,E2 -26674.21} C_VEL
LIN {X 0,Y 148.159,Z 711.001,A -85,B 0,C 180,E1 -26675.677,E2 -26675.677} C_VEL
LIN {X 0,Y 142.88,Z 722.203,A -85,B 0,C 180,E1 -26677.52,E2 -26677.52} C_VEL
LIN {X 0,Y 137.112,Z 732.299,A -85,B 0,C 180,E1 -26679.75,E2 -26679.75} C_VEL
LIN {X 0,Y 131.039,Z 741.411,A -85,B 0,C 180,E1 -26682.487,E2 -26682.487} C_VEL
LIN {X 0,Y 124.199,Z 750.303,A -85,B 0,C 180,E1 -26686.118,E2 -26686.118} C_VEL
LIN {X 0,Y 117.986,Z 757.466,A -85,B 0,C 180,E1 -26690.184,E2 -26690.184} C_VEL
LIN {X 0,Y 111.772,Z 764.006,A -85,B 0,C 180,E1 -26695.536,E2 -26695.536} C_VEL
LIN {X 0,Y 107.108,Z 768.344,A -85,B 0,C 180,E1 -26700.521,E2 -26700.521} C_VEL
LIN {X 0,Y 103.304,Z 771.623,A -85,B 0,C 180,E1 -26705.909,E2 -26705.909} C_VEL
LIN {X 0,Y 99.887,Z 774.511,A -85,B 0,C 180,E1 -26713.654,E2 -26713.654} C_VEL
LIN {X 0,Y 98.832,Z 775.339,A -85,B 0,C 180,E1 -26717.683,E2 -26717.683} C_VEL
LIN {X 0,Y 98.205,Z 775.752,A -85,B 0,C 180,E1 -26721.771,E2 -26721.771} C_VEL
LIN {X 0,Y 97.946,Z 775.782,A -85,B 0,C 180,E1 -26725.885,E2 -26725.885} C_VEL
LIN {X 0,Y 98.076,Z 775.428,A -85,B 0,C 180,E1 -26730,E2 -26730} C_VEL
LIN {X 0,Y 98.011,Z 774.653,A -85,B 0,C 180,E1 -26734.112,E2 -26734.112} C_VEL
LIN {X 0,Y 98.213,Z 773.434,A -85,B 0,C 180,E1 -26738.228,E2 -26738.228} C_VEL
LIN {X 0,Y 99.22,Z 770.839,A -85,B 0,C 180,E1 -26744.354,E2 -26744.354} C_VEL
LIN {X 0,Y 101.159,Z 767.223,A -85,B 0,C 180,E1 -26750.326,E2 -26750.326} C_VEL
LIN {X 0,Y 104.237,Z 762.497,A -85,B 0,C 180,E1 -26755.992,E2 -26755.992} C_VEL
LIN {X 0,Y 108.239,Z 756.515,A -85,B 0,C 180,E1 -26761.294,E2 -26761.294} C_VEL
LIN {X 0,Y 112.747,Z 749.321,A -85,B 0,C 180,E1 -26766.089,E2 -26766.089} C_VEL
LIN {X 0,Y 117.365,Z 741.433,A -85,B 0,C 180,E1 -26770.069,E2 -26770.069} C_VEL
LIN {X 0,Y 122.408,Z 732.217,A -85,B 0,C 180,E1 -26773.548,E2 -26773.548} C_VEL
LIN {X 0,Y 127.352,Z 721.965,A -85,B 0,C 180,E1 -26776.41,E2 -26776.41} C_VEL
LIN {X 0,Y 131.959,Z 710.58,A -85,B 0,C 180,E1 -26778.787,E2 -26778.787} C_VEL
LIN {X 0,Y 135.911,Z 698.755,A -85,B 0,C 180,E1 -26780.57,E2 -26780.57} C_VEL
LIN {X 0,Y 139.075,Z 686.086,A -85,B 0,C 180,E1 -26781.927,E2 -26781.927} C_VEL
LIN {X 0,Y 139.21,Z 685.539,A -85,B 0,C 180,E1 -26781.962,E2 -26781.962} C_VEL
LIN {X 0,Y 140.064,Z 679.872,A -85,B 0,C 180,E1 -26782.527,E2 -26782.527} C_VEL
LIN {X 0,Y 139.608,Z 670.64,A -85,B 0,C 180,E1 -26783.999,E2 -26783.999} C_VEL
LIN {X 0,Y 138.599,Z 661.317,A -85,B 0,C 180,E1 -26785.411,E2 -26785.411} C_VEL
LIN {X 0,Y 138.645,Z 655.487,A -85,B 0,C 180,E1 -26785.869,E2 -26785.869} C_VEL
LIN {X 0,Y 139.99,Z 639.533,A -85,B 0,C 180,E1 -26786.479,E2 -26786.479} C_VEL
LIN {X 0,Y 137.473,Z 631.638,A -85,B 0,C 180,E1 -26788.694,E2 -26788.694} C_VEL
LIN {X 0,Y 134.002,Z 622.581,A -85,B 0,C 180,E1 -26791.941,E2 -26791.941} C_VEL
LIN {X 0,Y 130.811,Z 617.07,A -85,B 0,C 180,E1 -26795.076,E2 -26795.076} C_VEL
LIN {X 0,Y 127.177,Z 611.134,A -85,B 0,C 180,E1 -26799.305,E2 -26799.305} C_VEL
LIN {X 0,Y 124.213,Z 606.708,A -85,B 0,C 180,E1 -26803.567,E2 -26803.567} C_VEL
LIN {X 0,Y 122.046,Z 603.427,A -85,B 0,C 180,E1 -26807.599,E2 -26807.599} C_VEL
LIN {X 0,Y 121.644,Z 602.498,A -85,B 0,C 180,E1 -26808.57,E2 -26808.57} C_VEL
LIN {X 0,Y 119.096,Z 598.937,A -85,B 0,C 180,E1 -26817.252,E2 -26817.252} C_VEL
LIN {X 0,Y 118.928,Z 597.396,A -85,B 0,C 180,E1 -26820,E2 -26820} C_VEL
LIN {X 0,Y 118.868,Z 597.474,A -85,B 0,C 180,E1 -26823.682,E2 -26823.682} C_VEL
LIN {X 0,Y 120.807,Z 602.017,A -85,B 0,C 180,E1 -26834.004,E2 -26834.004} C_VEL
LIN {X 0,Y 121.819,Z 602.976,A -85,B 0,C 180,E1 -26836.335,E2 -26836.335} C_VEL
LIN {X 0,Y 123.746,Z 606.301,A -85,B 0,C 180,E1 -26840.163,E2 -26840.163} C_VEL
LIN {X 0,Y 124.939,Z 607.788,A -85,B 0,C 180,E1 -26842.034,E2 -26842.034} C_VEL
LIN {X 0,Y 127.975,Z 612.506,A -85,B 0,C 180,E1 -26846.172,E2 -26846.172} C_VEL
LIN {X 0,Y 131.145,Z 617.576,A -85,B 0,C 180,E1 -26849.723,E2 -26849.723} C_VEL
LIN {X 0,Y 135.396,Z 625.215,A -85,B 0,C 180,E1 -26853.777,E2 -26853.777} C_VEL
LIN {X 0,Y 138.864,Z 632.315,A -85,B 0,C 180,E1 -26856.683,E2 -26856.683} C_VEL
LIN {X 0,Y 140.252,Z 635.337,A -85,B 0,C 180,E1 -26857.766,E2 -26857.766} C_VEL
LIN {X 0,Y 137.404,Z 667.437,A -85,B 0,C 180,E1 -26859.069,E2 -26859.069} C_VEL
LIN {X 0,Y 135.194,Z 680.44,A -85,B 0,C 180,E1 -26859.988,E2 -26859.988} C_VEL
LIN {X 0,Y 132.144,Z 692.87,A -85,B 0,C 180,E1 -26861.336,E2 -26861.336} C_VEL
LIN {X 0,Y 128.472,Z 703.956,A -85,B 0,C 180,E1 -26862.974,E2 -26862.974} C_VEL
LIN {X 0,Y 123.896,Z 715.513,A -85,B 0,C 180,E1 -26865.416,E2 -26865.416} C_VEL
LIN {X 0,Y 118.866,Z 725.92,A -85,B 0,C 180,E1 -26868.307,E2 -26868.307} C_VEL
LIN {X 0,Y 113.528,Z 735.308,A -85,B 0,C 180,E1 -26871.754,E2 -26871.754} C_VEL
LIN {X 0,Y 107.752,Z 744.341,A -85,B 0,C 180,E1 -26876.331,E2 -26876.331} C_VEL
LIN {X 0,Y 102.895,Z 751.61,A -85,B 0,C 180,E1 -26881.438,E2 -26881.438} C_VEL
LIN {X 0,Y 98.708,Z 757.444,A -85,B 0,C 180,E1 -26886.946,E2 -26886.946} C_VEL
LIN {X 0,Y 95.405,Z 762.046,A -85,B 0,C 180,E1 -26892.863,E2 -26892.863} C_VEL
LIN {X 0,Y 93.617,Z 764.502,A -85,B 0,C 180,E1 -26896.985,E2 -26896.985} C_VEL
LIN {X 0,Y 92.329,Z 766.494,A -85,B 0,C 180,E1 -26901.244,E2 -26901.244} C_VEL
LIN {X 0,Y 91.493,Z 768.076,A -85,B 0,C 180,E1 -26905.595,E2 -26905.595} C_VEL
LIN {X 0,Y 91.046,Z 769.258,A -85,B 0,C 180,E1 -26910,E2 -26910} C_VEL
LIN {X 0,Y 90.907,Z 770.007,A -85,B 0,C 180,E1 -26914.434,E2 -26914.434} C_VEL
LIN {X 0,Y 91.071,Z 770.373,A -85,B 0,C 180,E1 -26918.878,E2 -26918.878} C_VEL
LIN {X 0,Y 91.652,Z 770.36,A -85,B 0,C 180,E1 -26923.299,E2 -26923.299} C_VEL
LIN {X 0,Y 92.657,Z 769.962,A -85,B 0,C 180,E1 -26927.661,E2 -26927.661} C_VEL
LIN {X 0,Y 94.072,Z 769.131,A -85,B 0,C 180,E1 -26931.934,E2 -26931.934} C_VEL
LIN {X 0,Y 96.049,Z 767.895,A -85,B 0,C 180,E1 -26936.041,E2 -26936.041} C_VEL
LIN {X 0,Y 100.47,Z 764.695,A -85,B 0,C 180,E1 -26942.92,E2 -26942.92} C_VEL
LIN {X 0,Y 106.003,Z 760.176,A -85,B 0,C 180,E1 -26949.038,E2 -26949.038} C_VEL
LIN {X 0,Y 112.67,Z 753.979,A -85,B 0,C 180,E1 -26954.565,E2 -26954.565} C_VEL
LIN {X 0,Y 119.136,Z 747.215,A -85,B 0,C 180,E1 -26958.774,E2 -26958.774} C_VEL
LIN {X 0,Y 126.034,Z 738.776,A -85,B 0,C 180,E1 -26962.617,E2 -26962.617} C_VEL
LIN {X 0,Y 132.222,Z 730.063,A -85,B 0,C 180,E1 -26965.472,E2 -26965.472} C_VEL
LIN {X 0,Y 138.76,Z 719.318,A -85,B 0,C 180,E1 -26968.032,E2 -26968.032} C_VEL
LIN {X 0,Y 144.146,Z 708.576,A -85,B 0,C 180,E1 -26969.928,E2 -26969.928} C_VEL
LIN {X 0,Y 148.696,Z 697.044,A -85,B 0,C 180,E1 -26971.476,E2 -26971.476} C_VEL
LIN {X 0,Y 152.584,Z 684.297,A -85,B 0,C 180,E1 -26972.683,E2 -26972.683} C_VEL
LIN {X 0,Y 155.327,Z 671.403,A -85,B 0,C 180,E1 -26973.514,E2 -26973.514} C_VEL
LIN {X 0,Y 157.211,Z 655.935,A -85,B 0,C 180,E1 -26974.073,E2 -26974.073} C_VEL
LIN {X 0,Y 157.687,Z 650.511,A -85,B 0,C 180,E1 -26974.264,E2 -26974.264} C_VEL
LIN {X 0,Y 154.142,Z 642.977,A -85,B 0,C 180,E1 -26977.728,E2 -26977.728} C_VEL
LIN {X 0,Y 150.994,Z 636.927,A -85,B 0,C 180,E1 -26981.337,E2 -26981.337} C_VEL
LIN {X 0,Y 148.837,Z 633.121,A -85,B 0,C 180,E1 -26984.271,E2 -26984.271} C_VEL
LIN {X 0,Y 147.039,Z 629.948,A -85,B 0,C 180,E1 -26987.228,E2 -26987.228} C_VEL
LIN {X 0,Y 145.167,Z 626.414,A -85,B 0,C 180,E1 -26991.298,E2 -26991.298} C_VEL
LIN {X 0,Y 143.329,Z 622.265,A -85,B 0,C 180,E1 -26999.648,E2 -26999.648} C_VEL
LIN {X 0,Y 143.288,Z 621.93,A -85,B 0,C 180,E1 -27002.811,E2 -27002.811} C_VEL
LIN {X 0,Y 143.345,Z 622.641,A -85,B 0,C 180,E1 -27004.569,E2 -27004.569} C_VEL
LIN {X 0,Y 144.696,Z 626.106,A -85,B 0,C 180,E1 -27011.203,E2 -27011.203} C_VEL
LIN {X 0,Y 145.402,Z 627.001,A -85,B 0,C 180,E1 -27012.982,E2 -27012.982} C_VEL
LIN {X 0,Y 147.914,Z 631.51,A -85,B 0,C 180,E1 -27017.935,E2 -27017.935} C_VEL
LIN {X 0,Y 150.429,Z 635.922,A -85,B 0,C 180,E1 -27021.587,E2 -27021.587} C_VEL
LIN {X 0,Y 152.754,Z 641.479,A -85,B 0,C 180,E1 -27024.552,E2 -27024.552} C_VEL
LIN {X 0,Y 155.387,Z 648.723,A -85,B 0,C 180,E1 -27027.528,E2 -27027.528} C_VEL
LIN {X 0,Y 157.288,Z 654.627,A -85,B 0,C 180,E1 -27029.501,E2 -27029.501} C_VEL
LIN {X 0,Y 155.27,Z 673.586,A -85,B 0,C 180,E1 -27030.187,E2 -27030.187} C_VEL
LIN {X 0,Y 152.816,Z 685.94,A -85,B 0,C 180,E1 -27030.879,E2 -27030.879} C_VEL
LIN {X 0,Y 149.101,Z 698.772,A -85,B 0,C 180,E1 -27031.959,E2 -27031.959} C_VEL
LIN {X 0,Y 144.151,Z 711.23,A -85,B 0,C 180,E1 -27033.394,E2 -27033.394} C_VEL
LIN {X 0,Y 138.683,Z 722.351,A -85,B 0,C 180,E1 -27035.2,E2 -27035.2} C_VEL
LIN {X 0,Y 132.685,Z 732.361,A -85,B 0,C 180,E1 -27037.393,E2 -27037.393} C_VEL
LIN {X 0,Y 126.342,Z 741.429,A -85,B 0,C 180,E1 -27040.106,E2 -27040.106} C_VEL
LIN {X 0,Y 119.168,Z 750.284,A -85,B 0,C 180,E1 -27043.745,E2 -27043.745} C_VEL
LIN {X 0,Y 112.602,Z 757.406,A -85,B 0,C 180,E1 -27047.861,E2 -27047.861} C_VEL
LIN {X 0,Y 105.971,Z 763.911,A -85,B 0,C 180,E1 -27053.354,E2 -27053.354} C_VEL
LIN {X 0,Y 100.948,Z 768.223,A -85,B 0,C 180,E1 -27058.524,E2 -27058.524} C_VEL
LIN {X 0,Y 96.858,Z 771.479,A -85,B 0,C 180,E1 -27064.193,E2 -27064.193} C_VEL
LIN {X 0,Y 93.06,Z 774.344,A -85,B 0,C 180,E1 -27072.418,E2 -27072.418} C_VEL
LIN {X 0,Y 91.883,Z 775.15,A -85,B 0,C 180,E1 -27076.735,E2 -27076.735} C_VEL
LIN {X 0,Y 90.875,Z 775.572,A -85,B 0,C 180,E1 -27085.565,E2 -27085.565} C_VEL
LIN {X 0,Y 90.974,Z 775.207,A -85,B 0,C 180,E1 -27090,E2 -27090} C_VEL
LIN {X 0,Y 90.921,Z 774.411,A -85,B 0,C 180,E1 -27094.433,E2 -27094.433} C_VEL
LIN {X 0,Y 91.164,Z 773.179,A -85,B 0,C 180,E1 -27098.869,E2 -27098.869} C_VEL
LIN {X 0,Y 92.323,Z 770.56,A -85,B 0,C 180,E1 -27105.452,E2 -27105.452} C_VEL
LIN {X 0,Y 94.495,Z 766.918,A -85,B 0,C 180,E1 -27111.831,E2 -27111.831} C_VEL
LIN {X 0,Y 97.874,Z 762.167,A -85,B 0,C 180,E1 -27117.822,E2 -27117.822} C_VEL
LIN {X 0,Y 102.234,Z 756.157,A -85,B 0,C 180,E1 -27123.363,E2 -27123.363} C_VEL
LIN {X 0,Y 107.055,Z 748.928,A -85,B 0,C 180,E1 -27128.343,E2 -27128.343} C_VEL
LIN {X 0,Y 111.988,Z 741.002,A -85,B 0,C 180,E1 -27132.424,E2 -27132.424} C_VEL
LIN {X 0,Y 117.361,Z 731.733,A -85,B 0,C 180,E1 -27135.938,E2 -27135.938} C_VEL
LIN {X 0,Y 122.545,Z 721.404,A -85,B 0,C 180,E1 -27138.825,E2 -27138.825} C_VEL
LIN {X 0,Y 127.388,Z 709.94,A -85,B 0,C 180,E1 -27141.192,E2 -27141.192} C_VEL
LIN {X 0,Y 131.53,Z 697.987,A -85,B 0,C 180,E1 -27142.952,E2 -27142.952} C_VEL
LIN {X 0,Y 134.852,Z 684.969,A -85,B 0,C 180,E1 -27144.297,E2 -27144.297} C_VEL
LIN {X 0,Y 137.174,Z 671.328,A -85,B 0,C 180,E1 -27145.225,E2 -27145.225} C_VEL
LIN {X 0,Y 138.645,Z 655.487,A -85,B 0,C 180,E1 -27145.869,E2 -27145.869} C_VEL
LIN {X 0,Y 138.608,Z 651.643,A -85,B 0,C 180,E1 -27146.221,E2 -27146.221} C_VEL
LIN {X 0,Y 137.996,Z 648.056,A -85,B 0,C 180,E1 -27146.889,E2 -27146.889} C_VEL
LIN {X 0,Y 135.892,Z 641.526,A -85,B 0,C 180,E1 -27148.774,E2 -27148.774} C_VEL
LIN {X 0,Y 134.431,Z 637.266,A -85,B 0,C 180,E1 -27150.148,E2 -27150.148} C_VEL
LIN {X 0,Y 131.25,Z 628.21,A -85,B 0,C 180,E1 -27153.436,E2 -27153.436} C_VEL
LIN {X 0,Y 128.518,Z 623.116,A -85,B 0,C 180,E1 -27156.376,E2 -27156.376} C_VEL
LIN {X 0,Y 125.23,Z 617.43,A -85,B 0,C 180,E1 -27160.536,E2 -27160.536} C_VEL
LIN {X 0,Y 122.617,Z 613.274,A -85,B 0,C 180,E1 -27164.628,E2 -27164.628} C_VEL
LIN {X 0,Y 120.57,Z 609.808,A -85,B 0,C 180,E1 -27168.867,E2 -27168.867} C_VEL
LIN {X 0,Y 119.998,Z 608.975,A -85,B 0,C 180,E1 -27170.307,E2 -27170.307} C_VEL
LIN {X 0,Y 118.086,Z 605.537,A -85,B 0,C 180,E1 -27178.508,E2 -27178.508} C_VEL
LIN {X 0,Y 118.023,Z 604.754,A -85,B 0,C 180,E1 -27180,E2 -27180} C_VEL
LIN {X 0,Y 117.98,Z 604.709,A -85,B 0,C 180,E1 -27183.71,E2 -27183.71} C_VEL
LIN {X 0,Y 119.751,Z 608.981,A -85,B 0,C 180,E1 -27193.578,E2 -27193.578} C_VEL
LIN {X 0,Y 120.537,Z 609.859,A -85,B 0,C 180,E1 -27195.536,E2 -27195.536} C_VEL
LIN {X 0,Y 122.496,Z 613.248,A -85,B 0,C 180,E1 -27199.644,E2 -27199.644} C_VEL
LIN {X 0,Y 123.278,Z 614.345,A -85,B 0,C 180,E1 -27200.966,E2 -27200.966} C_VEL
LIN {X 0,Y 125.975,Z 618.772,A -85,B 0,C 180,E1 -27204.954,E2 -27204.954} C_VEL
LIN {X 0,Y 129.07,Z 624.017,A -85,B 0,C 180,E1 -27208.694,E2 -27208.694} C_VEL
LIN {X 0,Y 133.132,Z 631.849,A -85,B 0,C 180,E1 -27212.846,E2 -27212.846} C_VEL
LIN {X 0,Y 135.985,Z 638.223,A -85,B 0,C 180,E1 -27215.433,E2 -27215.433} C_VEL
LIN {X 0,Y 133.232,Z 667.818,A -85,B 0,C 180,E1 -27216.641,E2 -27216.641} C_VEL
LIN {X 0,Y 130.869,Z 681.077,A -85,B 0,C 180,E1 -27217.578,E2 -27217.578} C_VEL
LIN {X 0,Y 127.58,Z 693.73,A -85,B 0,C 180,E1 -27218.956,E2 -27218.956} C_VEL
LIN {X 0,Y 123.759,Z 704.626,A -85,B 0,C 180,E1 -27220.578,E2 -27220.578} C_VEL
LIN {X 0,Y 118.956,Z 716.097,A -85,B 0,C 180,E1 -27223.021,E2 -27223.021} C_VEL
LIN {X 0,Y 113.683,Z 726.439,A -85,B 0,C 180,E1 -27225.935,E2 -27225.935} C_VEL
LIN {X 0,Y 108.071,Z 735.755,A -85,B 0,C 180,E1 -27229.436,E2 -27229.436} C_VEL
LIN {X 0,Y 101.943,Z 744.745,A -85,B 0,C 180,E1 -27234.128,E2 -27234.128} C_VEL
LIN {X 0,Y 96.726,Z 751.979,A -85,B 0,C 180,E1 -27239.43,E2 -27239.43} C_VEL
LIN {X 0,Y 92.246,Z 757.781,A -85,B 0,C 180,E1 -27245.227,E2 -27245.227} C_VEL
LIN {X 0,Y 88.665,Z 762.355,A -85,B 0,C 180,E1 -27251.515,E2 -27251.515} C_VEL
LIN {X 0,Y 86.739,Z 764.784,A -85,B 0,C 180,E1 -27255.932,E2 -27255.932} C_VEL
LIN {X 0,Y 85.349,Z 766.764,A -85,B 0,C 180,E1 -27260.521,E2 -27260.521} C_VEL
LIN {X 0,Y 84.434,Z 768.334,A -85,B 0,C 180,E1 -27265.225,E2 -27265.225} C_VEL
LIN {X 0,Y 83.944,Z 769.497,A -85,B 0,C 180,E1 -27270,E2 -27270} C_VEL
LIN {X 0,Y 83.808,Z 770.23,A -85,B 0,C 180,E1 -27274.81,E2 -27274.81} C_VEL
LIN {X 0,Y 84.031,Z 770.584,A -85,B 0,C 180,E1 -27279.629,E2 -27279.629} C_VEL
LIN {X 0,Y 84.718,Z 770.56,A -85,B 0,C 180,E1 -27284.41,E2 -27284.41} C_VEL
LIN {X 0,Y 85.854,Z 770.145,A -85,B 0,C 180,E1 -27289.113,E2 -27289.113} C_VEL
LIN {X 0,Y 89.671,Z 768.048,A -85,B 0,C 180,E1 -27298.05,E2 -27298.05} C_VEL
LIN {X 0,Y 94.155,Z 765.08,A -85,B 0,C 180,E1 -27304.806,E2 -27304.806} C_VEL
LIN {X 0,Y 100.542,Z 760.263,A -85,B 0,C 180,E1 -27311.609,E2 -27311.609} C_VEL
LIN {X 0,Y 107.698,Z 754.036,A -85,B 0,C 180,E1 -27317.233,E2 -27317.233} C_VEL
LIN {X 0,Y 114.536,Z 747.239,A -85,B 0,C 180,E1 -27321.474,E2 -27321.474} C_VEL
LIN {X 0,Y 120.579,Z 740.289,A -85,B 0,C 180,E1 -27324.684,E2 -27324.684} C_VEL
LIN {X 0,Y 126.994,Z 731.903,A -85,B 0,C 180,E1 -27327.558,E2 -27327.558} C_VEL
LIN {X 0,Y 133.051,Z 722.708,A -85,B 0,C 180,E1 -27329.876,E2 -27329.876} C_VEL
LIN {X 0,Y 138.609,Z 712.675,A -85,B 0,C 180,E1 -27331.758,E2 -27331.758} C_VEL
LIN {X 0,Y 143.925,Z 700.679,A -85,B 0,C 180,E1 -27333.481,E2 -27333.481} C_VEL
LIN {X 0,Y 148.192,Z 688.241,A -85,B 0,C 180,E1 -27334.767,E2 -27334.767} C_VEL
LIN {X 0,Y 151.413,Z 675.004,A -85,B 0,C 180,E1 -27335.682,E2 -27335.682} C_VEL
LIN {X 0,Y 153.352,Z 662.572,A -85,B 0,C 180,E1 -27336.203,E2 -27336.203} C_VEL
LIN {X 0,Y 154.216,Z 653.951,A -85,B 0,C 180,E1 -27336.473,E2 -27336.473} C_VEL
LIN {X 0,Y 150.749,Z 646.356,A -85,B 0,C 180,E1 -27340.353,E2 -27340.353} C_VEL
LIN {X 0,Y 147.715,Z 640.291,A -85,B 0,C 180,E1 -27344.516,E2 -27344.516} C_VEL
LIN {X 0,Y 145.521,Z 636.364,A -85,B 0,C 180,E1 -27348.332,E2 -27348.332} C_VEL
LIN {X 0,Y 144.022,Z 633.259,A -85,B 0,C 180,E1 -27351.935,E2 -27351.935} C_VEL
LIN {X 0,Y 142.418,Z 629.061,A -85,B 0,C 180,E1 -27360.707,E2 -27360.707} C_VEL
LIN {X 0,Y 142.434,Z 629.042,A -85,B 0,C 180,E1 -27363.182,E2 -27363.182} C_VEL
LIN {X 0,Y 143.478,Z 632.805,A -85,B 0,C 180,E1 -27370.228,E2 -27370.228} C_VEL
LIN {X 0,Y 144.259,Z 633.921,A -85,B 0,C 180,E1 -27372.412,E2 -27372.412} C_VEL
LIN {X 0,Y 146.443,Z 638.121,A -85,B 0,C 180,E1 -27377.066,E2 -27377.066} C_VEL
LIN {X 0,Y 148.51,Z 641.947,A -85,B 0,C 180,E1 -27380.336,E2 -27380.336} C_VEL
LIN {X 0,Y 150.479,Z 647.028,A -85,B 0,C 180,E1 -27383.117,E2 -27383.117} C_VEL
LIN {X 0,Y 152.908,Z 654.342,A -85,B 0,C 180,E1 -27386.164,E2 -27386.164} C_VEL
LIN {X 0,Y 153.867,Z 657.507,A -85,B 0,C 180,E1 -27387.279,E2 -27387.279} C_VEL
LIN {X 0,Y 151.847,Z 674.699,A -85,B 0,C 180,E1 -27387.897,E2 -27387.897} C_VEL
LIN {X 0,Y 149.238,Z 686.843,A -85,B 0,C 180,E1 -27388.563,E2 -27388.563} C_VEL
LIN {X 0,Y 145.472,Z 699.118,A -85,B 0,C 180,E1 -27389.589,E2 -27389.589} C_VEL
LIN {X 0,Y 140.376,Z 711.463,A -85,B 0,C 180,E1 -27390.98,E2 -27390.98} C_VEL
LIN {X 0,Y 134.724,Z 722.493,A -85,B 0,C 180,E1 -27392.738,E2 -27392.738} C_VEL
LIN {X 0,Y 128.498,Z 732.426,A -85,B 0,C 180,E1 -27394.877,E2 -27394.877} C_VEL
LIN {X 0,Y 121.886,Z 741.449,A -85,B 0,C 180,E1 -27397.551,E2 -27397.551} C_VEL
LIN {X 0,Y 114.374,Z 750.266,A -85,B 0,C 180,E1 -27401.174,E2 -27401.174} C_VEL
LIN {X 0,Y 107.435,Z 757.343,A -85,B 0,C 180,E1 -27405.315,E2 -27405.315} C_VEL
LIN {X 0,Y 100.332,Z 763.816,A -85,B 0,C 180,E1 -27410.92,E2 -27410.92} C_VEL
LIN {X 0,Y 94.932,Z 768.102,A -85,B 0,C 180,E1 -27416.274,E2 -27416.274} C_VEL
LIN {X 0,Y 90.511,Z 771.336,A -85,B 0,C 180,E1 -27422.233,E2 -27422.233} C_VEL
LIN {X 0,Y 88.097,Z 772.953,A -85,B 0,C 180,E1 -27426.492,E2 -27426.492} C_VEL
LIN {X 0,Y 86.292,Z 774.175,A -85,B 0,C 180,E1 -27430.988,E2 -27430.988} C_VEL
LIN {X 0,Y 84.973,Z 774.961,A -85,B 0,C 180,E1 -27435.634,E2 -27435.634} C_VEL
LIN {X 0,Y 83.791,Z 775.361,A -85,B 0,C 180,E1 -27445.189,E2 -27445.189} C_VEL
LIN {X 0,Y 83.88,Z 774.986,A -85,B 0,C 180,E1 -27450,E2 -27450} C_VEL
LIN {X 0,Y 83.824,Z 774.167,A -85,B 0,C 180,E1 -27454.809,E2 -27454.809} C_VEL
LIN {X 0,Y 84.144,Z 772.924,A -85,B 0,C 180,E1 -27459.616,E2 -27459.616} C_VEL
LIN {X 0,Y 85.477,Z 770.281,A -85,B 0,C 180,E1 -27466.724,E2 -27466.724} C_VEL
LIN {X 0,Y 87.907,Z 766.615,A -85,B 0,C 180,E1 -27473.561,E2 -27473.561} C_VEL
LIN {X 0,Y 91.623,Z 761.837,A -85,B 0,C 180,E1 -27479.906,E2 -27479.906} C_VEL
LIN {X 0,Y 96.36,Z 755.798,A -85,B 0,C 180,E1 -27485.695,E2 -27485.695} C_VEL
LIN {X 0,Y 100.773,Z 749.627,A -85,B 0,C 180,E1 -27490.172,E2 -27490.172} C_VEL
LIN {X 0,Y 106.832,Z 740.573,A -85,B 0,C 180,E1 -27495.006,E2 -27495.006} C_VEL
LIN {X 0,Y 112.504,Z 731.238,A -85,B 0,C 180,E1 -27498.557,E2 -27498.557} C_VEL
LIN {X 0,Y 117.96,Z 720.841,A -85,B 0,C 180,E1 -27501.44,E2 -27501.44} C_VEL
LIN {X 0,Y 123.054,Z 709.3,A -85,B 0,C 180,E1 -27503.775,E2 -27503.775} C_VEL
LIN {X 0,Y 127.374,Z 697.174,A -85,B 0,C 180,E1 -27505.504,E2 -27505.504} C_VEL
LIN {X 0,Y 130.783,Z 684.132,A -85,B 0,C 180,E1 -27506.81,E2 -27506.81} C_VEL
LIN {X 0,Y 133.058,Z 671.052,A -85,B 0,C 180,E1 -27507.681,E2 -27507.681} C_VEL
LIN {X 0,Y 135.783,Z 641.668,A -85,B 0,C 180,E1 -27508.83,E2 -27508.83} C_VEL
LIN {X 0,Y 134.431,Z 637.266,A -85,B 0,C 180,E1 -27510.148,E2 -27510.148} C_VEL
LIN {X 0,Y 133.313,Z 634.437,A -85,B 0,C 180,E1 -27511.214,E2 -27511.214} C_VEL
LIN {X 0,Y 131.208,Z 631.142,A -85,B 0,C 180,E1 -27513.144,E2 -27513.144} C_VEL
LIN {X 0,Y 128.91,Z 628.735,A -85,B 0,C 180,E1 -27515.331,E2 -27515.331} C_VEL
LIN {X 0,Y 123.232,Z 623.569,A -85,B 0,C 180,E1 -27521.971,E2 -27521.971} C_VEL
LIN {X 0,Y 121,Z 619.72,A -85,B 0,C 180,E1 -27525.843,E2 -27525.843} C_VEL
LIN {X 0,Y 118.974,Z 615.946,A -85,B 0,C 180,E1 -27530.651,E2 -27530.651} C_VEL
LIN {X 0,Y 117.176,Z 612.639,A -85,B 0,C 180,E1 -27538.792,E2 -27538.792} C_VEL
LIN {X 0,Y 117.105,Z 611.739,A -85,B 0,C 180,E1 -27540.971,E2 -27540.971} C_VEL
LIN {X 0,Y 117.095,Z 612.068,A -85,B 0,C 180,E1 -27544.034,E2 -27544.034} C_VEL
LIN {X 0,Y 118.594,Z 615.853,A -85,B 0,C 180,E1 -27552.84,E2 -27552.84} C_VEL
LIN {X 0,Y 119.243,Z 616.622,A -85,B 0,C 180,E1 -27554.609,E2 -27554.609} C_VEL
LIN {X 0,Y 121.381,Z 620.328,A -85,B 0,C 180,E1 -27559.337,E2 -27559.337} C_VEL
LIN {X 0,Y 124.231,Z 625.395,A -85,B 0,C 180,E1 -27563.984,E2 -27563.984} C_VEL
LIN {X 0,Y 126.897,Z 630.314,A -85,B 0,C 180,E1 -27567.478,E2 -27567.478} C_VEL
LIN {X 0,Y 130.53,Z 637.776,A -85,B 0,C 180,E1 -27571.514,E2 -27571.514} C_VEL
LIN {X 0,Y 131.969,Z 641.15,A -85,B 0,C 180,E1 -27572.966,E2 -27572.966} C_VEL
LIN {X 0,Y 129.259,Z 668.656,A -85,B 0,C 180,E1 -27574.098,E2 -27574.098} C_VEL
LIN {X 0,Y 126.788,Z 681.749,A -85,B 0,C 180,E1 -27575.016,E2 -27575.016} C_VEL
LIN {X 0,Y 123.252,Z 694.546,A -85,B 0,C 180,E1 -27576.406,E2 -27576.406} C_VEL
LIN {X 0,Y 118.635,Z 706.865,A -85,B 0,C 180,E1 -27578.287,E2 -27578.287} C_VEL
LIN {X 0,Y 113.611,Z 717.964,A -85,B 0,C 180,E1 -27580.732,E2 -27580.732} C_VEL
LIN {X 0,Y 108.718,Z 726.954,A -85,B 0,C 180,E1 -27583.345,E2 -27583.345} C_VEL
LIN {X 0,Y 102.808,Z 736.196,A -85,B 0,C 180,E1 -27586.875,E2 -27586.875} C_VEL
LIN {X 0,Y 97.292,Z 743.803,A -85,B 0,C 180,E1 -27590.798,E2 -27590.798} C_VEL
LIN {X 0,Y 91.607,Z 751.237,A -85,B 0,C 180,E1 -27596.207,E2 -27596.207} C_VEL
LIN {X 0,Y 85.863,Z 758.116,A -85,B 0,C 180,E1 -27603.245,E2 -27603.245} C_VEL
LIN {X 0,Y 81.97,Z 762.66,A -85,B 0,C 180,E1 -27609.944,E2 -27609.944} C_VEL
LIN {X 0,Y 79.893,Z 765.066,A -85,B 0,C 180,E1 -27614.699,E2 -27614.699} C_VEL
LIN {X 0,Y 78.38,Z 767.033,A -85,B 0,C 180,E1 -27619.669,E2 -27619.669} C_VEL
LIN {X 0,Y 77.381,Z 768.591,A -85,B 0,C 180,E1 -27624.789,E2 -27624.789} C_VEL
LIN {X 0,Y 76.849,Z 769.733,A -85,B 0,C 180,E1 -27630,E2 -27630} C_VEL
LIN {X 0,Y 76.733,Z 770.452,A -85,B 0,C 180,E1 -27635.255,E2 -27635.255} C_VEL
LIN {X 0,Y 77.829,Z 770.759,A -85,B 0,C 180,E1 -27645.717,E2 -27645.717} C_VEL
LIN {X 0,Y 79.119,Z 770.326,A -85,B 0,C 180,E1 -27650.812,E2 -27650.812} C_VEL
LIN {X 0,Y 83.411,Z 768.201,A -85,B 0,C 180,E1 -27660.367,E2 -27660.367} C_VEL
LIN {X 0,Y 87.983,Z 765.453,A -85,B 0,C 180,E1 -27666.984,E2 -27666.984} C_VEL
LIN {X 0,Y 93.318,Z 761.815,A -85,B 0,C 180,E1 -27672.672,E2 -27672.672} C_VEL
LIN {X 0,Y 99.555,Z 756.979,A -85,B 0,C 180,E1 -27677.835,E2 -27677.835} C_VEL
LIN {X 0,Y 106.561,Z 750.865,A -85,B 0,C 180,E1 -27682.318,E2 -27682.318} C_VEL
LIN {X 0,Y 113.577,Z 743.672,A -85,B 0,C 180,E1 -27686.157,E2 -27686.157} C_VEL
LIN {X 0,Y 120.582,Z 735.416,A -85,B 0,C 180,E1 -27689.279,E2 -27689.279} C_VEL
LIN {X 0,Y 127.484,Z 725.839,A -85,B 0,C 180,E1 -27691.889,E2 -27691.889} C_VEL
LIN {X 0,Y 133.927,Z 715.193,A -85,B 0,C 180,E1 -27693.979,E2 -27693.979} C_VEL
LIN {X 0,Y 139.57,Z 703.556,A -85,B 0,C 180,E1 -27695.696,E2 -27695.696} C_VEL
LIN {X 0,Y 144.107,Z 691.474,A -85,B 0,C 180,E1 -27696.983,E2 -27696.983} C_VEL
LIN {X 0,Y 147.712,Z 678.494,A -85,B 0,C 180,E1 -27697.948,E2 -27697.948} C_VEL
LIN {X 0,Y 150.058,Z 665.581,A -85,B 0,C 180,E1 -27698.536,E2 -27698.536} C_VEL
LIN {X 0,Y 150.901,Z 657.394,A -85,B 0,C 180,E1 -27698.853,E2 -27698.853} C_VEL
LIN {X 0,Y 148.075,Z 651.003,A -85,B 0,C 180,E1 -27702.476,E2 -27702.476} C_VEL
LIN {X 0,Y 145.69,Z 646.018,A -85,B 0,C 180,E1 -27706.22,E2 -27706.22} C_VEL
LIN {X 0,Y 144.207,Z 643.021,A -85,B 0,C 180,E1 -27709.138,E2 -27709.138} C_VEL
LIN {X 0,Y 142.894,Z 640.118,A -85,B 0,C 180,E1 -27712.582,E2 -27712.582} C_VEL
LIN {X 0,Y 141.55,Z 636.119,A -85,B 0,C 180,E1 -27720.711,E2 -27720.711} C_VEL
LIN {X 0,Y 141.544,Z 636.293,A -85,B 0,C 180,E1 -27723.202,E2 -27723.202} C_VEL
LIN {X 0,Y 142.612,Z 639.965,A -85,B 0,C 180,E1 -27730.29,E2 -27730.29} C_VEL
LIN {X 0,Y 143.094,Z 640.748,A -85,B 0,C 180,E1 -27731.724,E2 -27731.724} C_VEL
LIN {X 0,Y 145.01,Z 644.713,A -85,B 0,C 180,E1 -27736.181,E2 -27736.181} C_VEL
LIN {X 0,Y 146.979,Z 648.685,A -85,B 0,C 180,E1 -27739.555,E2 -27739.555} C_VEL
LIN {X 0,Y 149.209,Z 655.433,A -85,B 0,C 180,E1 -27742.958,E2 -27742.958} C_VEL
LIN {X 0,Y 150.651,Z 660.394,A -85,B 0,C 180,E1 -27744.926,E2 -27744.926} C_VEL
LIN {X 0,Y 148.895,Z 674.422,A -85,B 0,C 180,E1 -27745.439,E2 -27745.439} C_VEL
LIN {X 0,Y 145.985,Z 687.387,A -85,B 0,C 180,E1 -27746.121,E2 -27746.121} C_VEL
LIN {X 0,Y 142.112,Z 699.464,A -85,B 0,C 180,E1 -27747.108,E2 -27747.108} C_VEL
LIN {X 0,Y 136.866,Z 711.697,A -85,B 0,C 180,E1 -27748.437,E2 -27748.437} C_VEL
LIN {X 0,Y 131.024,Z 722.622,A -85,B 0,C 180,E1 -27750.128,E2 -27750.128} C_VEL
LIN {X 0,Y 124.576,Z 732.492,A -85,B 0,C 180,E1 -27752.199,E2 -27752.199} C_VEL
LIN {X 0,Y 117.697,Z 741.47,A -85,B 0,C 180,E1 -27754.812,E2 -27754.812} C_VEL
LIN {X 0,Y 109.833,Z 750.248,A -85,B 0,C 180,E1 -27758.387,E2 -27758.387} C_VEL
LIN {X 0,Y 102.487,Z 757.277,A -85,B 0,C 180,E1 -27762.51,E2 -27762.51} C_VEL
LIN {X 0,Y 94.895,Z 763.723,A -85,B 0,C 180,E1 -27768.2,E2 -27768.2} C_VEL
LIN {X 0,Y 89.09,Z 767.983,A -85,B 0,C 180,E1 -27773.727,E2 -27773.727} C_VEL
LIN {X 0,Y 84.262,Z 771.192,A -85,B 0,C 180,E1 -27779.972,E2 -27779.972} C_VEL
LIN {X 0,Y 81.605,Z 772.798,A -85,B 0,C 180,E1 -27784.494,E2 -27784.494} C_VEL
LIN {X 0,Y 79.593,Z 774.004,A -85,B 0,C 180,E1 -27789.318,E2 -27789.318} C_VEL
LIN {X 0,Y 77.133,Z 775.153,A -85,B 0,C 180,E1 -27799.501,E2 -27799.501} C_VEL
LIN {X 0,Y 76.729,Z 775.151,A -85,B 0,C 180,E1 -27804.745,E2 -27804.745} C_VEL
LIN {X 0,Y 76.778,Z 774.763,A -85,B 0,C 180,E1 -27810,E2 -27810} C_VEL
LIN {X 0,Y 76.752,Z 773.923,A -85,B 0,C 180,E1 -27815.254,E2 -27815.254} C_VEL
LIN {X 0,Y 77.127,Z 772.669,A -85,B 0,C 180,E1 -27820.5,E2 -27820.5} C_VEL
LIN {X 0,Y 78.689,Z 770.003,A -85,B 0,C 180,E1 -27828.215,E2 -27828.215} C_VEL
LIN {X 0,Y 81.416,Z 766.31,A -85,B 0,C 180,E1 -27835.569,E2 -27835.569} C_VEL
LIN {X 0,Y 85.511,Z 761.506,A -85,B 0,C 180,E1 -27842.29,E2 -27842.29} C_VEL
LIN {X 0,Y 91.472,Z 754.395,A -85,B 0,C 180,E1 -27849.227,E2 -27849.227} C_VEL
LIN {X 0,Y 97.5,Z 746.428,A -85,B 0,C 180,E1 -27854.651,E2 -27854.651} C_VEL
LIN {X 0,Y 103.088,Z 738.389,A -85,B 0,C 180,E1 -27858.582,E2 -27858.582} C_VEL
LIN {X 0,Y 109.182,Z 728.586,A -85,B 0,C 180,E1 -27862.046,E2 -27862.046} C_VEL
LIN {X 0,Y 114.978,Z 717.665,A -85,B 0,C 180,E1 -27864.837,E2 -27864.837} C_VEL
LIN {X 0,Y 119.687,Z 706.966,A -85,B 0,C 180,E1 -27866.797,E2 -27866.797} C_VEL
LIN {X 0,Y 123.817,Z 695.202,A -85,B 0,C 180,E1 -27868.364,E2 -27868.364} C_VEL
LIN {X 0,Y 127.271,Z 681.951,A -85,B 0,C 180,E1 -27869.597,E2 -27869.597} C_VEL
LIN {X 0,Y 129.383,Z 669.309,A -85,B 0,C 180,E1 -27870.353,E2 -27870.353} C_VEL
LIN {X 0,Y 131.8,Z 643.969,A -85,B 0,C 180,E1 -27871.321,E2 -27871.321} C_VEL
LIN {X 0,Y 129.008,Z 635.104,A -85,B 0,C 180,E1 -27874.488,E2 -27874.488} C_VEL
LIN {X 0,Y 127.724,Z 631.864,A -85,B 0,C 180,E1 -27876.008,E2 -27876.008} C_VEL
LIN {X 0,Y 124.365,Z 625.612,A -85,B 0,C 180,E1 -27880.288,E2 -27880.288} C_VEL
LIN {X 0,Y 123.232,Z 623.569,A -85,B 0,C 180,E1 -27881.971,E2 -27881.971} C_VEL
LIN {X 0,Y 121.55,Z 622.036,A -85,B 0,C 180,E1 -27884.535,E2 -27884.535} C_VEL
LIN {X 0,Y 118.984,Z 621.435,A -85,B 0,C 180,E1 -27889.109,E2 -27889.109} C_VEL
LIN {X 0,Y 116.856,Z 621.283,A -85,B 0,C 180,E1 -27894.899,E2 -27894.899} C_VEL
LIN {X 0,Y 116.48,Z 620.755,A -85,B 0,C 180,E1 -27896.848,E2 -27896.848} C_VEL
LIN {X 0,Y 116.233,Z 618.828,A -85,B 0,C 180,E1 -27900.978,E2 -27900.978} C_VEL
LIN {X 0,Y 116.21,Z 619.023,A -85,B 0,C 180,E1 -27903.468,E2 -27903.468} C_VEL
LIN {X 0,Y 117.595,Z 622.852,A -85,B 0,C 180,E1 -27912.513,E2 -27912.513} C_VEL
LIN {X 0,Y 118.018,Z 623.484,A -85,B 0,C 180,E1 -27913.781,E2 -27913.781} C_VEL
LIN {X 0,Y 120.235,Z 627.716,A -85,B 0,C 180,E1 -27919.03,E2 -27919.03} C_VEL
LIN {X 0,Y 122.467,Z 631.895,A -85,B 0,C 180,E1 -27922.896,E2 -27922.896} C_VEL
LIN {X 0,Y 124.987,Z 637.021,A -85,B 0,C 180,E1 -27926.486,E2 -27926.486} C_VEL
LIN {X 0,Y 128.052,Z 643.811,A -85,B 0,C 180,E1 -27930.184,E2 -27930.184} C_VEL
LIN {X 0,Y 128.196,Z 644.221,A -85,B 0,C 180,E1 -27930.353,E2 -27930.353} C_VEL
LIN {X 0,Y 125.693,Z 668.524,A -85,B 0,C 180,E1 -27931.335,E2 -27931.335} C_VEL
LIN {X 0,Y 123.075,Z 681.964,A -85,B 0,C 180,E1 -27932.246,E2 -27932.246} C_VEL
LIN {X 0,Y 119.815,Z 693.537,A -85,B 0,C 180,E1 -27933.448,E2 -27933.448} C_VEL
LIN {X 0,Y 115.777,Z 704.373,A -85,B 0,C 180,E1 -27934.968,E2 -27934.968} C_VEL
LIN {X 0,Y 110.448,Z 715.975,A -85,B 0,C 180,E1 -27937.309,E2 -27937.309} C_VEL
LIN {X 0,Y 104.65,Z 726.403,A -85,B 0,C 180,E1 -27940.192,E2 -27940.192} C_VEL
LIN {X 0,Y 98.934,Z 734.948,A -85,B 0,C 180,E1 -27943.271,E2 -27943.271} C_VEL
LIN {X 0,Y 93.015,Z 742.816,A -85,B 0,C 180,E1 -27947.156,E2 -27947.156} C_VEL
LIN {X 0,Y 86.773,Z 750.497,A -85,B 0,C 180,E1 -27952.596,E2 -27952.596} C_VEL
LIN {X 0,Y 81.234,Z 756.658,A -85,B 0,C 180,E1 -27958.729,E2 -27958.729} C_VEL
LIN {X 0,Y 76.689,Z 761.555,A -85,B 0,C 180,E1 -27965.646,E2 -27965.646} C_VEL
LIN {X 0,Y 73.078,Z 765.348,A -85,B 0,C 180,E1 -27973.231,E2 -27973.231} C_VEL
LIN {X 0,Y 71.429,Z 767.302,A -85,B 0,C 180,E1 -27978.651,E2 -27978.651} C_VEL
LIN {X 0,Y 70.321,Z 768.849,A -85,B 0,C 180,E1 -27984.264,E2 -27984.264} C_VEL
LIN {X 0,Y 69.746,Z 769.967,A -85,B 0,C 180,E1 -27990,E2 -27990} C_VEL
LIN {X 0,Y 69.636,Z 770.675,A -85,B 0,C 180,E1 -27995.792,E2 -27995.792} C_VEL
LIN {X 0,Y 70.019,Z 771.007,A -85,B 0,C 180,E1 -28001.58,E2 -28001.58} C_VEL
LIN {X 0,Y 70.978,Z 770.959,A -85,B 0,C 180,E1 -28007.28,E2 -28007.28} C_VEL
LIN {X 0,Y 72.47,Z 770.503,A -85,B 0,C 180,E1 -28012.824,E2 -28012.824} C_VEL
LIN {X 0,Y 77.311,Z 768.354,A -85,B 0,C 180,E1 -28023.054,E2 -28023.054} C_VEL
LIN {X 0,Y 81.89,Z 765.858,A -85,B 0,C 180,E1 -28029.429,E2 -28029.429} C_VEL
LIN {X 0,Y 88.181,Z 761.916,A -85,B 0,C 180,E1 -28035.83,E2 -28035.83} C_VEL
LIN {X 0,Y 94.893,Z 757.052,A -85,B 0,C 180,E1 -28041.045,E2 -28041.045} C_VEL
LIN {X 0,Y 102.338,Z 750.906,A -85,B 0,C 180,E1 -28045.494,E2 -28045.494} C_VEL
LIN {X 0,Y 110.196,Z 743.213,A -85,B 0,C 180,E1 -28049.455,E2 -28049.455} C_VEL
LIN {X 0,Y 117.086,Z 735.36,A -85,B 0,C 180,E1 -28052.293,E2 -28052.293} C_VEL
LIN {X 0,Y 124.282,Z 725.73,A -85,B 0,C 180,E1 -28054.791,E2 -28054.791} C_VEL
LIN {X 0,Y 130.962,Z 715.018,A -85,B 0,C 180,E1 -28056.778,E2 -28056.778} C_VEL
LIN {X 0,Y 136.729,Z 703.381,A -85,B 0,C 180,E1 -28058.404,E2 -28058.404} C_VEL
LIN {X 0,Y 141.498,Z 690.922,A -85,B 0,C 180,E1 -28059.654,E2 -28059.654} C_VEL
LIN {X 0,Y 145.231,Z 677.577,A -85,B 0,C 180,E1 -28060.558,E2 -28060.558} C_VEL
LIN {X 0,Y 147.471,Z 664.982,A -85,B 0,C 180,E1 -28061.088,E2 -28061.088} C_VEL
LIN {X 0,Y 147.905,Z 661.18,A -85,B 0,C 180,E1 -28061.241,E2 -28061.241} C_VEL
LIN {X 0,Y 145.583,Z 655.581,A -85,B 0,C 180,E1 -28064.724,E2 -28064.724} C_VEL
LIN {X 0,Y 143.822,Z 651.706,A -85,B 0,C 180,E1 -28067.942,E2 -28067.942} C_VEL
LIN {X 0,Y 142.826,Z 649.527,A -85,B 0,C 180,E1 -28070.178,E2 -28070.178} C_VEL
LIN {X 0,Y 141.678,Z 646.798,A -85,B 0,C 180,E1 -28073.591,E2 -28073.591} C_VEL
LIN {X 0,Y 140.667,Z 643.101,A -85,B 0,C 180,E1 -28081.574,E2 -28081.574} C_VEL
LIN {X 0,Y 140.66,Z 643.344,A -85,B 0,C 180,E1 -28082.864,E2 -28082.864} C_VEL
LIN {X 0,Y 141.638,Z 646.964,A -85,B 0,C 180,E1 -28090.001,E2 -28090.001} C_VEL
LIN {X 0,Y 142.241,Z 648.359,A -85,B 0,C 180,E1 -28091.941,E2 -28091.941} C_VEL
LIN {X 0,Y 143.6,Z 651.271,A -85,B 0,C 180,E1 -28095.251,E2 -28095.251} C_VEL
LIN {X 0,Y 145.225,Z 654.853,A -85,B 0,C 180,E1 -28098.334,E2 -28098.334} C_VEL
LIN {X 0,Y 147.094,Z 661.192,A -85,B 0,C 180,E1 -28101.549,E2 -28101.549} C_VEL
LIN {X 0,Y 147.679,Z 663.452,A -85,B 0,C 180,E1 -28102.479,E2 -28102.479} C_VEL
LIN {X 0,Y 145.786,Z 676.511,A -85,B 0,C 180,E1 -28102.983,E2 -28102.983} C_VEL
LIN {X 0,Y 142.302,Z 690.29,A -85,B 0,C 180,E1 -28103.734,E2 -28103.734} C_VEL
LIN {X 0,Y 138.263,Z 701.792,A -85,B 0,C 180,E1 -28104.691,E2 -28104.691} C_VEL
LIN {X 0,Y 132.878,Z 713.411,A -85,B 0,C 180,E1 -28105.958,E2 -28105.958} C_VEL
LIN {X 0,Y 126.87,Z 723.916,A -85,B 0,C 180,E1 -28107.588,E2 -28107.588} C_VEL
LIN {X 0,Y 119.515,Z 734.507,A -85,B 0,C 180,E1 -28109.848,E2 -28109.848} C_VEL
LIN {X 0,Y 112.396,Z 743.113,A -85,B 0,C 180,E1 -28112.422,E2 -28112.422} C_VEL
LIN {X 0,Y 104.227,Z 751.475,A -85,B 0,C 180,E1 -28115.988,E2 -28115.988} C_VEL
LIN {X 0,Y 96.592,Z 758.222,A -85,B 0,C 180,E1 -28120.185,E2 -28120.185} C_VEL
LIN {X 0,Y 89.696,Z 763.629,A -85,B 0,C 180,E1 -28125.157,E2 -28125.157} C_VEL
LIN {X 0,Y 83.454,Z 767.864,A -85,B 0,C 180,E1 -28130.833,E2 -28130.833} C_VEL
LIN {X 0,Y 78.172,Z 771.048,A -85,B 0,C 180,E1 -28137.356,E2 -28137.356} C_VEL
LIN {X 0,Y 75.228,Z 772.642,A -85,B 0,C 180,E1 -28142.154,E2 -28142.154} C_VEL
LIN {X 0,Y 72.961,Z 773.83,A -85,B 0,C 180,E1 -28147.338,E2 -28147.338} C_VEL
LIN {X 0,Y 70.153,Z 774.953,A -85,B 0,C 180,E1 -28158.442,E2 -28158.442} C_VEL
LIN {X 0,Y 69.643,Z 774.94,A -85,B 0,C 180,E1 -28164.208,E2 -28164.208} C_VEL
LIN {X 0,Y 69.699,Z 774.539,A -85,B 0,C 180,E1 -28170,E2 -28170} C_VEL
LIN {X 0,Y 69.662,Z 773.679,A -85,B 0,C 180,E1 -28175.79,E2 -28175.79} C_VEL
LIN {X 0,Y 70.144,Z 772.413,A -85,B 0,C 180,E1 -28181.559,E2 -28181.559} C_VEL
LIN {X 0,Y 71.945,Z 769.723,A -85,B 0,C 180,E1 -28189.992,E2 -28189.992} C_VEL
LIN {X 0,Y 75.05,Z 766.006,A -85,B 0,C 180,E1 -28197.918,E2 -28197.918} C_VEL
LIN {X 0,Y 79.559,Z 761.174,A -85,B 0,C 180,E1 -28205.042,E2 -28205.042} C_VEL
LIN {X 0,Y 85.142,Z 755.074,A -85,B 0,C 180,E1 -28211.326,E2 -28211.326} C_VEL
LIN {X 0,Y 91.437,Z 747.474,A -85,B 0,C 180,E1 -28216.9,E2 -28216.9} C_VEL
LIN {X 0,Y 97.269,Z 739.706,A -85,B 0,C 180,E1 -28220.959,E2 -28220.959} C_VEL
LIN {X 0,Y 104.294,Z 729.158,A -85,B 0,C 180,E1 -28224.79,E2 -28224.79} C_VEL
LIN {X 0,Y 110.346,Z 718.416,A -85,B 0,C 180,E1 -28227.552,E2 -28227.552} C_VEL
LIN {X 0,Y 115.225,Z 708.008,A -85,B 0,C 180,E1 -28229.487,E2 -28229.487} C_VEL
LIN {X 0,Y 119.874,Z 695.502,A -85,B 0,C 180,E1 -28231.132,E2 -28231.132} C_VEL
LIN {X 0,Y 123.435,Z 682.47,A -85,B 0,C 180,E1 -28232.329,E2 -28232.329} C_VEL
LIN {X 0,Y 125.734,Z 669.748,A -85,B 0,C 180,E1 -28233.078,E2 -28233.078} C_VEL
LIN {X 0,Y 128.056,Z 646.495,A -85,B 0,C 180,E1 -28233.957,E2 -28233.957} C_VEL
LIN {X 0,Y 125.773,Z 638.63,A -85,B 0,C 180,E1 -28236.974,E2 -28236.974} C_VEL
LIN {X 0,Y 123.029,Z 632.927,A -85,B 0,C 180,E1 -28240.716,E2 -28240.716} C_VEL
LIN {X 0,Y 120.893,Z 628.965,A -85,B 0,C 180,E1 -28244.187,E2 -28244.187} C_VEL
LIN {X 0,Y 119.462,Z 626.221,A -85,B 0,C 180,E1 -28247.039,E2 -28247.039} C_VEL
LIN {X 0,Y 117.798,Z 622.821,A -85,B 0,C 180,E1 -28251.423,E2 -28251.423} C_VEL
LIN {X 0,Y 116.48,Z 620.755,A -85,B 0,C 180,E1 -28256.848,E2 -28256.848} C_VEL
LIN {X 0,Y 116.208,Z 620.531,A -85,B 0,C 180,E1 -28258.764,E2 -28258.764} C_VEL
LIN {X 0,Y 115.968,Z 621.111,A -85,B 0,C 180,E1 -28260.675,E2 -28260.675} C_VEL
LIN {X 0,Y 115.681,Z 623.77,A -85,B 0,C 180,E1 -28264.389,E2 -28264.389} C_VEL
LIN {X 0,Y 116.054,Z 628.695,A -85,B 0,C 180,E1 -28269.993,E2 -28269.993} C_VEL
LIN {X 0,Y 116.525,Z 629.753,A -85,B 0,C 180,E1 -28271.93,E2 -28271.93} C_VEL
LIN {X 0,Y 118.66,Z 634.142,A -85,B 0,C 180,E1 -28277.783,E2 -28277.783} C_VEL
LIN {X 0,Y 120.818,Z 638.572,A -85,B 0,C 180,E1 -28281.9,E2 -28281.9} C_VEL
LIN {X 0,Y 123.033,Z 643.542,A -85,B 0,C 180,E1 -28285.347,E2 -28285.347} C_VEL
LIN {X 0,Y 124.682,Z 647.495,A -85,B 0,C 180,E1 -28287.592,E2 -28287.592} C_VEL
LIN {X 0,Y 122.308,Z 669.292,A -85,B 0,C 180,E1 -28288.479,E2 -28288.479} C_VEL
LIN {X 0,Y 119.734,Z 681.918,A -85,B 0,C 180,E1 -28289.295,E2 -28289.295} C_VEL
LIN {X 0,Y 116.047,Z 694.439,A -85,B 0,C 180,E1 -28290.55,E2 -28290.55} C_VEL
LIN {X 0,Y 111.878,Z 705.043,A -85,B 0,C 180,E1 -28292.002,E2 -28292.002} C_VEL
LIN {X 0,Y 106.317,Z 716.555,A -85,B 0,C 180,E1 -28294.281,E2 -28294.281} C_VEL
LIN {X 0,Y 100.228,Z 726.92,A -85,B 0,C 180,E1 -28297.099,E2 -28297.099} C_VEL
LIN {X 0,Y 94.224,Z 735.412,A -85,B 0,C 180,E1 -28300.136,E2 -28300.136} C_VEL
LIN {X 0,Y 87.965,Z 743.236,A -85,B 0,C 180,E1 -28304.025,E2 -28304.025} C_VEL
LIN {X 0,Y 81.258,Z 750.864,A -85,B 0,C 180,E1 -28309.56,E2 -28309.56} C_VEL
LIN {X 0,Y 75.276,Z 756.993,A -85,B 0,C 180,E1 -28315.933,E2 -28315.933} C_VEL
LIN {X 0,Y 70.295,Z 761.863,A -85,B 0,C 180,E1 -28323.263,E2 -28323.263} C_VEL
LIN {X 0,Y 66.33,Z 765.63,A -85,B 0,C 180,E1 -28331.467,E2 -28331.467} C_VEL
LIN {X 0,Y 64.493,Z 767.572,A -85,B 0,C 180,E1 -28337.412,E2 -28337.412} C_VEL
LIN {X 0,Y 63.261,Z 769.106,A -85,B 0,C 180,E1 -28343.622,E2 -28343.622} C_VEL
LIN {X 0,Y 62.641,Z 770.201,A -85,B 0,C 180,E1 -28350,E2 -28350} C_VEL
LIN {X 0,Y 62.558,Z 770.898,A -85,B 0,C 180,E1 -28356.45,E2 -28356.45} C_VEL
LIN {X 0,Y 63.059,Z 771.218,A -85,B 0,C 180,E1 -28362.879,E2 -28362.879} C_VEL
LIN {X 0,Y 64.174,Z 771.16,A -85,B 0,C 180,E1 -28369.18,E2 -28369.18} C_VEL
LIN {X 0,Y 65.931,Z 770.68,A -85,B 0,C 180,E1 -28375.238,E2 -28375.238} C_VEL
LIN {X 0,Y 71.409,Z 768.507,A -85,B 0,C 180,E1 -28386.193,E2 -28386.193} C_VEL
LIN {X 0,Y 75.994,Z 766.252,A -85,B 0,C 180,E1 -28392.28,E2 -28392.28} C_VEL
LIN {X 0,Y 83.354,Z 762.017,A -85,B 0,C 180,E1 -28399.36,E2 -28399.36} C_VEL
LIN {X 0,Y 90.567,Z 757.125,A -85,B 0,C 180,E1 -28404.566,E2 -28404.566} C_VEL
LIN {X 0,Y 98.462,Z 750.948,A -85,B 0,C 180,E1 -28408.927,E2 -28408.927} C_VEL
LIN {X 0,Y 106.431,Z 743.521,A -85,B 0,C 180,E1 -28412.639,E2 -28412.639} C_VEL
LIN {X 0,Y 113.942,Z 735.305,A -85,B 0,C 180,E1 -28415.473,E2 -28415.473} C_VEL
LIN {X 0,Y 121.422,Z 725.624,A -85,B 0,C 180,E1 -28417.83,E2 -28417.83} C_VEL
LIN {X 0,Y 128.321,Z 714.848,A -85,B 0,C 180,E1 -28419.701,E2 -28419.701} C_VEL
LIN {X 0,Y 134.205,Z 703.219,A -85,B 0,C 180,E1 -28421.219,E2 -28421.219} C_VEL
LIN {X 0,Y 138.771,Z 691.665,A -85,B 0,C 180,E1 -28422.309,E2 -28422.309} C_VEL
LIN {X 0,Y 142.5,Z 678.932,A -85,B 0,C 180,E1 -28423.156,E2 -28423.156} C_VEL
LIN {X 0,Y 144.855,Z 666.965,A -85,B 0,C 180,E1 -28423.648,E2 -28423.648} C_VEL
LIN {X 0,Y 145.034,Z 664.866,A -85,B 0,C 180,E1 -28423.826,E2 -28423.826} C_VEL
LIN {X 0,Y 143,Z 659.52,A -85,B 0,C 180,E1 -28427.673,E2 -28427.673} C_VEL
LIN {X 0,Y 141.557,Z 656.137,A -85,B 0,C 180,E1 -28431.074,E2 -28431.074} C_VEL
LIN {X 0,Y 140.599,Z 653.645,A -85,B 0,C 180,E1 -28434.262,E2 -28434.262} C_VEL
LIN {X 0,Y 139.798,Z 650.17,A -85,B 0,C 180,E1 -28441.584,E2 -28441.584} C_VEL
LIN {X 0,Y 139.77,Z 650.662,A -85,B 0,C 180,E1 -28443.062,E2 -28443.062} C_VEL
LIN {X 0,Y 140.859,Z 654.472,A -85,B 0,C 180,E1 -28450.42,E2 -28450.42} C_VEL
LIN {X 0,Y 142.378,Z 658.197,A -85,B 0,C 180,E1 -28454.654,E2 -28454.654} C_VEL
LIN {X 0,Y 143.623,Z 661.304,A -85,B 0,C 180,E1 -28457.257,E2 -28457.257} C_VEL
LIN {X 0,Y 144.929,Z 666.608,A -85,B 0,C 180,E1 -28459.94,E2 -28459.94} C_VEL
LIN {X 0,Y 142.764,Z 679.186,A -85,B 0,C 180,E1 -28460.449,E2 -28460.449} C_VEL
LIN {X 0,Y 139.428,Z 691.42,A -85,B 0,C 180,E1 -28461.124,E2 -28461.124} C_VEL
LIN {X 0,Y 134.673,Z 703.915,A -85,B 0,C 180,E1 -28462.138,E2 -28462.138} C_VEL
LIN {X 0,Y 129.145,Z 715.029,A -85,B 0,C 180,E1 -28463.32,E2 -28463.32} C_VEL
LIN {X 0,Y 122.195,Z 726.375,A -85,B 0,C 180,E1 -28465.065,E2 -28465.065} C_VEL
LIN {X 0,Y 114.649,Z 736.396,A -85,B 0,C 180,E1 -28467.273,E2 -28467.273} C_VEL
LIN {X 0,Y 105.865,Z 746.098,A -85,B 0,C 180,E1 -28470.344,E2 -28470.344} C_VEL
LIN {X 0,Y 97.48,Z 753.862,A -85,B 0,C 180,E1 -28473.995,E2 -28473.995} C_VEL
LIN {X 0,Y 89.609,Z 760.093,A -85,B 0,C 180,E1 -28478.346,E2 -28478.346} C_VEL
LIN {X 0,Y 82.499,Z 765.063,A -85,B 0,C 180,E1 -28483.607,E2 -28483.607} C_VEL
LIN {X 0,Y 76.009,Z 768.912,A -85,B 0,C 180,E1 -28489.667,E2 -28489.667} C_VEL
LIN {X 0,Y 72.276,Z 770.905,A -85,B 0,C 180,E1 -28494.309,E2 -28494.309} C_VEL
LIN {X 0,Y 69.004,Z 772.487,A -85,B 0,C 180,E1 -28499.387,E2 -28499.387} C_VEL
LIN {X 0,Y 66.441,Z 773.654,A -85,B 0,C 180,E1 -28504.97,E2 -28504.97} C_VEL
LIN {X 0,Y 63.189,Z 774.753,A -85,B 0,C 180,E1 -28517.148,E2 -28517.148} C_VEL
LIN {X 0,Y 62.573,Z 774.73,A -85,B 0,C 180,E1 -28523.551,E2 -28523.551} C_VEL
LIN {X 0,Y 62.609,Z 774.312,A -85,B 0,C 180,E1 -28530,E2 -28530} C_VEL
LIN {X 0,Y 62.586,Z 773.435,A -85,B 0,C 180,E1 -28536.447,E2 -28536.447} C_VEL
LIN {X 0,Y 63.178,Z 772.157,A -85,B 0,C 180,E1 -28542.855,E2 -28542.855} C_VEL
LIN {X 0,Y 65.27,Z 769.443,A -85,B 0,C 180,E1 -28552.139,E2 -28552.139} C_VEL
LIN {X 0,Y 68.839,Z 765.702,A -85,B 0,C 180,E1 -28560.694,E2 -28560.694} C_VEL
LIN {X 0,Y 73.815,Z 760.841,A -85,B 0,C 180,E1 -28568.233,E2 -28568.233} C_VEL
LIN {X 0,Y 79.866,Z 754.709,A -85,B 0,C 180,E1 -28574.746,E2 -28574.746} C_VEL
LIN {X 0,Y 86.7,Z 747.076,A -85,B 0,C 180,E1 -28580.359,E2 -28580.359} C_VEL
LIN {X 0,Y 92.949,Z 739.267,A -85,B 0,C 180,E1 -28584.37,E2 -28584.37} C_VEL
LIN {X 0,Y 100.354,Z 728.655,A -85,B 0,C 180,E1 -28588.116,E2 -28588.116} C_VEL
LIN {X 0,Y 106.689,Z 717.851,A -85,B 0,C 180,E1 -28590.786,E2 -28590.786} C_VEL
LIN {X 0,Y 111.778,Z 707.339,A -85,B 0,C 180,E1 -28592.633,E2 -28592.633} C_VEL
LIN {X 0,Y 116.606,Z 694.668,A -85,B 0,C 180,E1 -28594.195,E2 -28594.195} C_VEL
LIN {X 0,Y 120.239,Z 681.644,A -85,B 0,C 180,E1 -28595.316,E2 -28595.316} C_VEL
LIN {X 0,Y 122.554,Z 668.768,A -85,B 0,C 180,E1 -28596.02,E2 -28596.02} C_VEL
LIN {X 0,Y 124.596,Z 649.048,A -85,B 0,C 180,E1 -28596.744,E2 -28596.744} C_VEL
LIN {X 0,Y 122.979,Z 643.269,A -85,B 0,C 180,E1 -28599.21,E2 -28599.21} C_VEL
LIN {X 0,Y 120.304,Z 637.475,A -85,B 0,C 180,E1 -28603.454,E2 -28603.454} C_VEL
LIN {X 0,Y 118.089,Z 632.897,A -85,B 0,C 180,E1 -28608.005,E2 -28608.005} C_VEL
LIN {X 0,Y 116.531,Z 629.553,A -85,B 0,C 180,E1 -28612.583,E2 -28612.583} C_VEL
LIN {X 0,Y 115.35,Z 625.802,A -85,B 0,C 180,E1 -28621.97,E2 -28621.97} C_VEL
LIN {X 0,Y 115.474,Z 627.688,A -85,B 0,C 180,E1 -28626.737,E2 -28626.737} C_VEL
LIN {X 0,Y 116.525,Z 629.753,A -85,B 0,C 180,E1 -28631.93,E2 -28631.93} C_VEL
LIN {X 0,Y 117.057,Z 630.973,A -85,B 0,C 180,E1 -28633.727,E2 -28633.727} C_VEL
LIN {X 0,Y 117.54,Z 632.938,A -85,B 0,C 180,E1 -28635.365,E2 -28635.365} C_VEL
LIN {X 0,Y 118.41,Z 638.183,A -85,B 0,C 180,E1 -28638.239,E2 -28638.239} C_VEL
LIN {X 0,Y 120.038,Z 647.008,A -85,B 0,C 180,E1 -28642.325,E2 -28642.325} C_VEL
LIN {X 0,Y 120.904,Z 649.5,A -85,B 0,C 180,E1 -28643.818,E2 -28643.818} C_VEL
LIN {X 0,Y 121.461,Z 650.842,A -85,B 0,C 180,E1 -28644.678,E2 -28644.678} C_VEL
LIN {X 0,Y 119.297,Z 669.641,A -85,B 0,C 180,E1 -28645.436,E2 -28645.436} C_VEL
LIN {X 0,Y 116.652,Z 682.141,A -85,B 0,C 180,E1 -28646.195,E2 -28646.195} C_VEL
LIN {X 0,Y 113.239,Z 693.514,A -85,B 0,C 180,E1 -28647.272,E2 -28647.272} C_VEL
LIN {X 0,Y 108.301,Z 705.703,A -85,B 0,C 180,E1 -28648.832,E2 -28648.832} C_VEL
LIN {X 0,Y 102.506,Z 717.131,A -85,B 0,C 180,E1 -28651.019,E2 -28651.019} C_VEL
LIN {X 0,Y 96.129,Z 727.433,A -85,B 0,C 180,E1 -28653.736,E2 -28653.736} C_VEL
LIN {X 0,Y 89.827,Z 735.874,A -85,B 0,C 180,E1 -28656.685,E2 -28656.685} C_VEL
LIN {X 0,Y 81.963,Z 745.006,A -85,B 0,C 180,E1 -28661.387,E2 -28661.387} C_VEL
LIN {X 0,Y 74.887,Z 752.338,A -85,B 0,C 180,E1 -28667.126,E2 -28667.126} C_VEL
LIN {X 0,Y 67.586,Z 759.096,A -85,B 0,C 180,E1 -28675.116,E2 -28675.116} C_VEL
LIN {X 0,Y 62.446,Z 763.555,A -85,B 0,C 180,E1 -28683.245,E2 -28683.245} C_VEL
LIN {X 0,Y 59.662,Z 765.912,A -85,B 0,C 180,E1 -28689.306,E2 -28689.306} C_VEL
LIN {X 0,Y 57.603,Z 767.841,A -85,B 0,C 180,E1 -28695.877,E2 -28695.877} C_VEL
LIN {X 0,Y 56.238,Z 769.36,A -85,B 0,C 180,E1 -28702.821,E2 -28702.821} C_VEL
LIN {X 0,Y 55.53,Z 770.435,A -85,B 0,C 180,E1 -28710,E2 -28710} C_VEL
LIN {X 0,Y 55.506,Z 771.121,A -85,B 0,C 180,E1 -28717.274,E2 -28717.274} C_VEL
LIN {X 0,Y 56.115,Z 771.43,A -85,B 0,C 180,E1 -28724.506,E2 -28724.506} C_VEL
LIN {X 0,Y 57.468,Z 771.358,A -85,B 0,C 180,E1 -28731.523,E2 -28731.523} C_VEL
LIN {X 0,Y 59.534,Z 770.857,A -85,B 0,C 180,E1 -28738.177,E2 -28738.177} C_VEL
LIN {X 0,Y 65.763,Z 768.66,A -85,B 0,C 180,E1 -28749.881,E2 -28749.881} C_VEL
LIN {X 0,Y 70.305,Z 766.652,A -85,B 0,C 180,E1 -28755.591,E2 -28755.591} C_VEL
LIN {X 0,Y 78.864,Z 762.12,A -85,B 0,C 180,E1 -28763.323,E2 -28763.323} C_VEL
LIN {X 0,Y 86.609,Z 757.199,A -85,B 0,C 180,E1 -28768.432,E2 -28768.432} C_VEL
LIN {X 0,Y 94.97,Z 750.992,A -85,B 0,C 180,E1 -28772.623,E2 -28772.623} C_VEL
LIN {X 0,Y 103.633,Z 743.219,A -85,B 0,C 180,E1 -28776.272,E2 -28776.272} C_VEL
LIN {X 0,Y 111.168,Z 735.252,A -85,B 0,C 180,E1 -28778.823,E2 -28778.823} C_VEL
LIN {X 0,Y 118.915,Z 725.52,A -85,B 0,C 180,E1 -28781.013,E2 -28781.013} C_VEL
LIN {X 0,Y 126.026,Z 714.673,A -85,B 0,C 180,E1 -28782.741,E2 -28782.741} C_VEL
LIN {X 0,Y 131.572,Z 704.039,A -85,B 0,C 180,E1 -28784.04,E2 -28784.04} C_VEL
LIN {X 0,Y 136.29,Z 692.578,A -85,B 0,C 180,E1 -28785.058,E2 -28785.058} C_VEL
LIN {X 0,Y 140.289,Z 679.438,A -85,B 0,C 180,E1 -28785.875,E2 -28785.875} C_VEL
LIN {X 0,Y 142.415,Z 669.024,A -85,B 0,C 180,E1 -28786.351,E2 -28786.351} C_VEL
LIN {X 0,Y 141.114,Z 665.059,A -85,B 0,C 180,E1 -28789.598,E2 -28789.598} C_VEL
LIN {X 0,Y 140.125,Z 662.267,A -85,B 0,C 180,E1 -28792.615,E2 -28792.615} C_VEL
LIN {X 0,Y 139.541,Z 660.485,A -85,B 0,C 180,E1 -28794.943,E2 -28794.943} C_VEL
LIN {X 0,Y 138.916,Z 657.364,A -85,B 0,C 180,E1 -28801.449,E2 -28801.449} C_VEL
LIN {X 0,Y 138.887,Z 657.785,A -85,B 0,C 180,E1 -28802.9,E2 -28802.9} C_VEL
LIN {X 0,Y 139.774,Z 661.342,A -85,B 0,C 180,E1 -28809.77,E2 -28809.77} C_VEL
LIN {X 0,Y 141.016,Z 664.733,A -85,B 0,C 180,E1 -28813.693,E2 -28813.693} C_VEL
LIN {X 0,Y 141.927,Z 667.442,A -85,B 0,C 180,E1 -28815.988,E2 -28815.988} C_VEL
LIN {X 0,Y 142.431,Z 669.948,A -85,B 0,C 180,E1 -28817.355,E2 -28817.355} C_VEL
LIN {X 0,Y 139.679,Z 683.061,A -85,B 0,C 180,E1 -28817.901,E2 -28817.901} C_VEL
LIN {X 0,Y 135.817,Z 695.316,A -85,B 0,C 180,E1 -28818.597,E2 -28818.597} C_VEL
LIN {X 0,Y 130.525,Z 707.671,A -85,B 0,C 180,E1 -28819.568,E2 -28819.568} C_VEL
LIN {X 0,Y 124.102,Z 719.258,A -85,B 0,C 180,E1 -28820.871,E2 -28820.871} C_VEL
LIN {X 0,Y 117.022,Z 729.689,A -85,B 0,C 180,E1 -28822.579,E2 -28822.579} C_VEL
LIN {X 0,Y 110.044,Z 738.223,A -85,B 0,C 180,E1 -28824.487,E2 -28824.487} C_VEL
LIN {X 0,Y 102.461,Z 746.103,A -85,B 0,C 180,E1 -28826.915,E2 -28826.915} C_VEL
LIN {X 0,Y 93.689,Z 753.814,A -85,B 0,C 180,E1 -28830.385,E2 -28830.385} C_VEL
LIN {X 0,Y 85.369,Z 760.014,A -85,B 0,C 180,E1 -28834.591,E2 -28834.591} C_VEL
LIN {X 0,Y 77.755,Z 764.957,A -85,B 0,C 180,E1 -28839.802,E2 -28839.802} C_VEL
LIN {X 0,Y 70.722,Z 768.781,A -85,B 0,C 180,E1 -28845.925,E2 -28845.925} C_VEL
LIN {X 0,Y 66.62,Z 770.761,A -85,B 0,C 180,E1 -28850.732,E2 -28850.732} C_VEL
LIN {X 0,Y 62.977,Z 772.332,A -85,B 0,C 180,E1 -28856.084,E2 -28856.084} C_VEL
LIN {X 0,Y 60.042,Z 773.476,A -85,B 0,C 180,E1 -28862.083,E2 -28862.083} C_VEL
LIN {X 0,Y 56.277,Z 774.554,A -85,B 0,C 180,E1 -28875.537,E2 -28875.537} C_VEL
LIN {X 0,Y 55.527,Z 774.52,A -85,B 0,C 180,E1 -28882.729,E2 -28882.729} C_VEL
LIN {X 0,Y 55.508,Z 774.082,A -85,B 0,C 180,E1 -28890,E2 -28890} C_VEL
LIN {X 0,Y 55.536,Z 773.191,A -85,B 0,C 180,E1 -28897.27,E2 -28897.27} C_VEL
LIN {X 0,Y 56.264,Z 771.902,A -85,B 0,C 180,E1 -28904.467,E2 -28904.467} C_VEL
LIN {X 0,Y 58.715,Z 769.162,A -85,B 0,C 180,E1 -28914.767,E2 -28914.767} C_VEL
LIN {X 0,Y 62.825,Z 765.398,A -85,B 0,C 180,E1 -28924.008,E2 -28924.008} C_VEL
LIN {X 0,Y 68.344,Z 760.509,A -85,B 0,C 180,E1 -28931.943,E2 -28931.943} C_VEL
LIN {X 0,Y 73.83,Z 755.475,A -85,B 0,C 180,E1 -28937.537,E2 -28937.537} C_VEL
LIN {X 0,Y 81.061,Z 748.049,A -85,B 0,C 180,E1 -28943.318,E2 -28943.318} C_VEL
LIN {X 0,Y 87.605,Z 740.481,A -85,B 0,C 180,E1 -28947.387,E2 -28947.387} C_VEL
LIN {X 0,Y 94.602,Z 731.326,A -85,B 0,C 180,E1 -28950.796,E2 -28950.796} C_VEL
LIN {X 0,Y 101.159,Z 721.175,A -85,B 0,C 180,E1 -28953.439,E2 -28953.439} C_VEL
LIN {X 0,Y 107.159,Z 709.893,A -85,B 0,C 180,E1 -28955.5,E2 -28955.5} C_VEL
LIN {X 0,Y 112.542,Z 697.206,A -85,B 0,C 180,E1 -28957.085,E2 -28957.085} C_VEL
LIN {X 0,Y 116.405,Z 684.765,A -85,B 0,C 180,E1 -28958.165,E2 -28958.165} C_VEL
LIN {X 0,Y 119.172,Z 671.567,A -85,B 0,C 180,E1 -28958.94,E2 -28958.94} C_VEL
LIN {X 0,Y 121.431,Z 651.728,A -85,B 0,C 180,E1 -28959.681,E2 -28959.681} C_VEL
LIN {X 0,Y 120.503,Z 648.33,A -85,B 0,C 180,E1 -28961.318,E2 -28961.318} C_VEL
LIN {X 0,Y 118.185,Z 642.757,A -85,B 0,C 180,E1 -28965.622,E2 -28965.622} C_VEL
LIN {X 0,Y 116.526,Z 639.191,A -85,B 0,C 180,E1 -28969.576,E2 -28969.576} C_VEL
LIN {X 0,Y 115.399,Z 636.379,A -85,B 0,C 180,E1 -28973.443,E2 -28973.443} C_VEL
LIN {X 0,Y 114.472,Z 633.017,A -85,B 0,C 180,E1 -28981.489,E2 -28981.489} C_VEL
LIN {X 0,Y 114.445,Z 633.323,A -85,B 0,C 180,E1 -28983.267,E2 -28983.267} C_VEL
LIN {X 0,Y 115.396,Z 636.598,A -85,B 0,C 180,E1 -28991.091,E2 -28991.091} C_VEL
LIN {X 0,Y 117.222,Z 640.766,A -85,B 0,C 180,E1 -28996.704,E2 -28996.704} C_VEL
LIN {X 0,Y 119.301,Z 645.387,A -85,B 0,C 180,E1 -29001.038,E2 -29001.038} C_VEL
LIN {X 0,Y 120.904,Z 649.5,A -85,B 0,C 180,E1 -29003.818,E2 -29003.818} C_VEL
LIN {X 0,Y 121.151,Z 651.354,A -85,B 0,C 180,E1 -29004.392,E2 -29004.392} C_VEL
LIN {X 0,Y 120.96,Z 653.692,A -85,B 0,C 180,E1 -29004.517,E2 -29004.517} C_VEL
LIN {X 0,Y 120.157,Z 657.469,A -85,B 0,C 180,E1 -29004.151,E2 -29004.151} C_VEL
LIN {X 0,Y 117.454,Z 666.375,A -85,B 0,C 180,E1 -29002.395,E2 -29002.395} C_VEL
LIN {X 0,Y 116.617,Z 670.109,A -85,B 0,C 180,E1 -29002.248,E2 -29002.248} C_VEL
LIN {X 0,Y 113.873,Z 682.612,A -85,B 0,C 180,E1 -29002.967,E2 -29002.967} C_VEL
LIN {X 0,Y 110.128,Z 694.512,A -85,B 0,C 180,E1 -29004.025,E2 -29004.025} C_VEL
LIN {X 0,Y 105.078,Z 706.36,A -85,B 0,C 180,E1 -29005.458,E2 -29005.458} C_VEL
LIN {X 0,Y 99.052,Z 717.705,A -85,B 0,C 180,E1 -29007.516,E2 -29007.516} C_VEL
LIN {X 0,Y 92.391,Z 727.941,A -85,B 0,C 180,E1 -29010.088,E2 -29010.088} C_VEL
LIN {X 0,Y 84.412,Z 737.955,A -85,B 0,C 180,E1 -29013.637,E2 -29013.637} C_VEL
LIN {X 0,Y 77.463,Z 745.404,A -85,B 0,C 180,E1 -29017.454,E2 -29017.454} C_VEL
LIN {X 0,Y 69.86,Z 752.703,A -85,B 0,C 180,E1 -29023.169,E2 -29023.169} C_VEL
LIN {X 0,Y 61.9,Z 759.416,A -85,B 0,C 180,E1 -29031.359,E2 -29031.359} C_VEL
LIN {X 0,Y 56.203,Z 763.849,A -85,B 0,C 180,E1 -29039.988,E2 -29039.988} C_VEL
LIN {X 0,Y 53.099,Z 766.193,A -85,B 0,C 180,E1 -29046.605,E2 -29046.605} C_VEL
LIN {X 0,Y 50.769,Z 768.109,A -85,B 0,C 180,E1 -29053.927,E2 -29053.927} C_VEL
LIN {X 0,Y 49.201,Z 769.611,A -85,B 0,C 180,E1 -29061.788,E2 -29061.788} C_VEL
LIN {X 0,Y 48.44,Z 770.669,A -85,B 0,C 180,E1 -29070,E2 -29070} C_VEL
LIN {X 0,Y 48.436,Z 771.344,A -85,B 0,C 180,E1 -29078.343,E2 -29078.343} C_VEL
LIN {X 0,Y 49.24,Z 771.642,A -85,B 0,C 180,E1 -29086.586,E2 -29086.586} C_VEL
LIN {X 0,Y 50.892,Z 771.554,A -85,B 0,C 180,E1 -29094.474,E2 -29094.474} C_VEL
LIN {X 0,Y 56.594,Z 770.12,A -85,B 0,C 180,E1 -29108.381,E2 -29108.381} C_VEL
LIN {X 0,Y 60.441,Z 768.814,A -85,B 0,C 180,E1 -29114.239,E2 -29114.239} C_VEL
LIN {X 0,Y 66.948,Z 766.139,A -85,B 0,C 180,E1 -29121.449,E2 -29121.449} C_VEL
LIN {X 0,Y 74.81,Z 762.223,A -85,B 0,C 180,E1 -29127.723,E2 -29127.723} C_VEL
LIN {X 0,Y 83.09,Z 757.274,A -85,B 0,C 180,E1 -29132.635,E2 -29132.635} C_VEL
LIN {X 0,Y 91.904,Z 751.036,A -85,B 0,C 180,E1 -29136.583,E2 -29136.583} C_VEL
LIN {X 0,Y 99.429,Z 744.641,A -85,B 0,C 180,E1 -29139.478,E2 -29139.478} C_VEL
LIN {X 0,Y 107.212,Z 736.952,A -85,B 0,C 180,E1 -29141.895,E2 -29141.895} C_VEL
LIN {X 0,Y 115.171,Z 727.559,A -85,B 0,C 180,E1 -29143.962,E2 -29143.962} C_VEL
LIN {X 0,Y 122.455,Z 717.101,A -85,B 0,C 180,E1 -29145.574,E2 -29145.574} C_VEL
LIN {X 0,Y 128.979,Z 705.453,A -85,B 0,C 180,E1 -29146.9,E2 -29146.9} C_VEL
LIN {X 0,Y 134.128,Z 693.504,A -85,B 0,C 180,E1 -29147.901,E2 -29147.901} C_VEL
LIN {X 0,Y 138.2,Z 680.707,A -85,B 0,C 180,E1 -29148.634,E2 -29148.634} C_VEL
LIN {X 0,Y 139.918,Z 673.233,A -85,B 0,C 180,E1 -29149.032,E2 -29149.032} C_VEL
LIN {X 0,Y 138.936,Z 669.482,A -85,B 0,C 180,E1 -29152.734,E2 -29152.734} C_VEL
LIN {X 0,Y 138.397,Z 667.309,A -85,B 0,C 180,E1 -29155.631,E2 -29155.631} C_VEL
LIN {X 0,Y 137.998,Z 664.555,A -85,B 0,C 180,E1 -29161.459,E2 -29161.459} C_VEL
LIN {X 0,Y 137.954,Z 665.104,A -85,B 0,C 180,E1 -29163.103,E2 -29163.103} C_VEL
LIN {X 0,Y 138.606,Z 668.19,A -85,B 0,C 180,E1 -29169.117,E2 -29169.117} C_VEL
LIN {X 0,Y 139.468,Z 671.277,A -85,B 0,C 180,E1 -29172.736,E2 -29172.736} C_VEL
LIN {X 0,Y 140.034,Z 673.402,A -85,B 0,C 180,E1 -29174.635,E2 -29174.635} C_VEL
LIN {X 0,Y 137.195,Z 685.423,A -85,B 0,C 180,E1 -29175.153,E2 -29175.153} C_VEL
LIN {X 0,Y 133.209,Z 697.106,A -85,B 0,C 180,E1 -29175.812,E2 -29175.812} C_VEL
LIN {X 0,Y 127.486,Z 709.494,A -85,B 0,C 180,E1 -29176.701,E2 -29176.701} C_VEL
LIN {X 0,Y 120.952,Z 720.707,A -85,B 0,C 180,E1 -29177.925,E2 -29177.925} C_VEL
LIN {X 0,Y 113.691,Z 730.814,A -85,B 0,C 180,E1 -29179.494,E2 -29179.494} C_VEL
LIN {X 0,Y 105.693,Z 739.934,A -85,B 0,C 180,E1 -29181.425,E2 -29181.425} C_VEL
LIN {X 0,Y 96.361,Z 748.831,A -85,B 0,C 180,E1 -29184.265,E2 -29184.265} C_VEL
LIN {X 0,Y 87.338,Z 755.999,A -85,B 0,C 180,E1 -29187.732,E2 -29187.732} C_VEL
LIN {X 0,Y 78.747,Z 761.732,A -85,B 0,C 180,E1 -29192.028,E2 -29192.028} C_VEL
LIN {X 0,Y 70.802,Z 766.26,A -85,B 0,C 180,E1 -29197.432,E2 -29197.432} C_VEL
LIN {X 0,Y 65.791,Z 768.651,A -85,B 0,C 180,E1 -29201.605,E2 -29201.605} C_VEL
LIN {X 0,Y 61.273,Z 770.619,A -85,B 0,C 180,E1 -29206.514,E2 -29206.514} C_VEL
LIN {X 0,Y 57.207,Z 772.178,A -85,B 0,C 180,E1 -29212.103,E2 -29212.103} C_VEL
LIN {X 0,Y 51.227,Z 774.017,A -85,B 0,C 180,E1 -29225.696,E2 -29225.696} C_VEL
LIN {X 0,Y 49.433,Z 774.355,A -85,B 0,C 180,E1 -29233.481,E2 -29233.481} C_VEL
LIN {X 0,Y 48.484,Z 774.309,A -85,B 0,C 180,E1 -29241.666,E2 -29241.666} C_VEL
LIN {X 0,Y 48.425,Z 773.85,A -85,B 0,C 180,E1 -29250,E2 -29250} C_VEL
LIN {X 0,Y 48.49,Z 772.947,A -85,B 0,C 180,E1 -29258.333,E2 -29258.333} C_VEL
LIN {X 0,Y 49.384,Z 771.645,A -85,B 0,C 180,E1 -29266.536,E2 -29266.536} C_VEL
LIN {X 0,Y 52.322,Z 768.882,A -85,B 0,C 180,E1 -29278.042,E2 -29278.042} C_VEL
LIN {X 0,Y 57.066,Z 765.093,A -85,B 0,C 180,E1 -29288.008,E2 -29288.008} C_VEL
LIN {X 0,Y 63.218,Z 760.176,A -85,B 0,C 180,E1 -29296.269,E2 -29296.269} C_VEL
LIN {X 0,Y 69.174,Z 755.108,A -85,B 0,C 180,E1 -29301.94,E2 -29301.94} C_VEL
LIN {X 0,Y 76.994,Z 747.65,A -85,B 0,C 180,E1 -29307.599,E2 -29307.599} C_VEL
LIN {X 0,Y 83.982,Z 740.046,A -85,B 0,C 180,E1 -29311.481,E2 -29311.481} C_VEL
LIN {X 0,Y 91.346,Z 730.843,A -85,B 0,C 180,E1 -29314.689,E2 -29314.689} C_VEL
LIN {X 0,Y 98.175,Z 720.603,A -85,B 0,C 180,E1 -29317.169,E2 -29317.169} C_VEL
LIN {X 0,Y 104.413,Z 709.242,A -85,B 0,C 180,E1 -29319.051,E2 -29319.051} C_VEL
LIN {X 0,Y 109.57,Z 697.444,A -85,B 0,C 180,E1 -29320.4,E2 -29320.4} C_VEL
LIN {X 0,Y 113.457,Z 685.542,A -85,B 0,C 180,E1 -29321.387,E2 -29321.387} C_VEL
LIN {X 0,Y 116.489,Z 671.845,A -85,B 0,C 180,E1 -29322.133,E2 -29322.133} C_VEL
LIN {X 0,Y 118.584,Z 654.537,A -85,B 0,C 180,E1 -29322.763,E2 -29322.763} C_VEL
LIN {X 0,Y 116.509,Z 648.944,A -85,B 0,C 180,E1 -29327.148,E2 -29327.148} C_VEL
LIN {X 0,Y 115.254,Z 645.881,A -85,B 0,C 180,E1 -29330.568,E2 -29330.568} C_VEL
LIN {X 0,Y 114.311,Z 643.19,A -85,B 0,C 180,E1 -29334.267,E2 -29334.267} C_VEL
LIN {X 0,Y 113.578,Z 640.294,A -85,B 0,C 180,E1 -29341.501,E2 -29341.501} C_VEL
LIN {X 0,Y 113.569,Z 640.34,A -85,B 0,C 180,E1 -29342.78,E2 -29342.78} C_VEL
LIN {X 0,Y 114.506,Z 643.972,A -85,B 0,C 180,E1 -29351.179,E2 -29351.179} C_VEL
LIN {X 0,Y 115.89,Z 647.565,A -85,B 0,C 180,E1 -29355.773,E2 -29355.773} C_VEL
LIN {X 0,Y 117.504,Z 651.525,A -85,B 0,C 180,E1 -29359.547,E2 -29359.547} C_VEL
LIN {X 0,Y 118.53,Z 654.532,A -85,B 0,C 180,E1 -29361.621,E2 -29361.621} C_VEL
LIN {X 0,Y 116.617,Z 670.109,A -85,B 0,C 180,E1 -29362.248,E2 -29362.248} C_VEL
LIN {X 0,Y 115.302,Z 675.866,A -85,B 0,C 180,E1 -29362.245,E2 -29362.245} C_VEL
LIN {X 0,Y 112.011,Z 685.102,A -85,B 0,C 180,E1 -29361.498,E2 -29361.498} C_VEL
LIN {X 0,Y 108.097,Z 694.136,A -85,B 0,C 180,E1 -29360.814,E2 -29360.814} C_VEL
LIN {X 0,Y 105.722,Z 699.536,A -85,B 0,C 180,E1 -29361.002,E2 -29361.002} C_VEL
LIN {X 0,Y 100.649,Z 710.142,A -85,B 0,C 180,E1 -29362.304,E2 -29362.304} C_VEL
LIN {X 0,Y 93.651,Z 721.89,A -85,B 0,C 180,E1 -29364.51,E2 -29364.51} C_VEL
LIN {X 0,Y 86.758,Z 731.36,A -85,B 0,C 180,E1 -29366.994,E2 -29366.994} C_VEL
LIN {X 0,Y 79.179,Z 740.017,A -85,B 0,C 180,E1 -29370.072,E2 -29370.072} C_VEL
LIN {X 0,Y 71.993,Z 747.146,A -85,B 0,C 180,E1 -29373.926,E2 -29373.926} C_VEL
LIN {X 0,Y 63.915,Z 754.145,A -85,B 0,C 180,E1 -29379.674,E2 -29379.674} C_VEL
LIN {X 0,Y 56.541,Z 759.736,A -85,B 0,C 180,E1 -29386.872,E2 -29386.872} C_VEL
LIN {X 0,Y 50.203,Z 764.142,A -85,B 0,C 180,E1 -29395.948,E2 -29395.948} C_VEL
LIN {X 0,Y 46.674,Z 766.474,A -85,B 0,C 180,E1 -29403.146,E2 -29403.146} C_VEL
LIN {X 0,Y 44.01,Z 768.378,A -85,B 0,C 180,E1 -29411.375,E2 -29411.375} C_VEL
LIN {X 0,Y 42.201,Z 769.859,A -85,B 0,C 180,E1 -29420.414,E2 -29420.414} C_VEL
LIN {X 0,Y 41.333,Z 770.902,A -85,B 0,C 180,E1 -29430,E2 -29430} C_VEL
LIN {X 0,Y 41.406,Z 771.566,A -85,B 0,C 180,E1 -29439.772,E2 -29439.772} C_VEL
LIN {X 0,Y 42.462,Z 771.853,A -85,B 0,C 180,E1 -29449.331,E2 -29449.331} C_VEL
LIN {X 0,Y 44.478,Z 771.747,A -85,B 0,C 180,E1 -29458.296,E2 -29458.296} C_VEL
LIN {X 0,Y 51.183,Z 770.285,A -85,B 0,C 180,E1 -29473.356,E2 -29473.356} C_VEL
LIN {X 0,Y 59.838,Z 767.436,A -85,B 0,C 180,E1 -29484.037,E2 -29484.037} C_VEL
LIN {X 0,Y 68.421,Z 763.744,A -85,B 0,C 180,E1 -29490.817,E2 -29490.817} C_VEL
LIN {X 0,Y 77.059,Z 759.156,A -85,B 0,C 180,E1 -29495.784,E2 -29495.784} C_VEL
LIN {X 0,Y 87.745,Z 752.196,A -85,B 0,C 180,E1 -29500.238,E2 -29500.238} C_VEL
LIN {X 0,Y 97.151,Z 744.651,A -85,B 0,C 180,E1 -29503.435,E2 -29503.435} C_VEL
LIN {X 0,Y 105.209,Z 736.918,A -85,B 0,C 180,E1 -29505.6,E2 -29505.6} C_VEL
LIN {X 0,Y 113.412,Z 727.455,A -85,B 0,C 180,E1 -29507.418,E2 -29507.418} C_VEL
LIN {X 0,Y 120.878,Z 716.932,A -85,B 0,C 180,E1 -29508.847,E2 -29508.847} C_VEL
LIN {X 0,Y 127.551,Z 705.187,A -85,B 0,C 180,E1 -29510.024,E2 -29510.024} C_VEL
LIN {X 0,Y 132.778,Z 693.158,A -85,B 0,C 180,E1 -29510.906,E2 -29510.906} C_VEL
LIN {X 0,Y 136.969,Z 680.038,A -85,B 0,C 180,E1 -29511.563,E2 -29511.563} C_VEL
LIN {X 0,Y 137.518,Z 677.824,A -85,B 0,C 180,E1 -29511.68,E2 -29511.68} C_VEL
LIN {X 0,Y 137,Z 674.328,A -85,B 0,C 180,E1 -29515.771,E2 -29515.771} C_VEL
LIN {X 0,Y 136.8,Z 671.712,A -85,B 0,C 180,E1 -29521.472,E2 -29521.472} C_VEL
LIN {X 0,Y 136.715,Z 672.43,A -85,B 0,C 180,E1 -29523.315,E2 -29523.315} C_VEL
LIN {X 0,Y 137.107,Z 674.977,A -85,B 0,C 180,E1 -29528.474,E2 -29528.474} C_VEL
LIN {X 0,Y 137.656,Z 677.896,A -85,B 0,C 180,E1 -29531.94,E2 -29531.94} C_VEL
LIN {X 0,Y 134.148,Z 690.247,A -85,B 0,C 180,E1 -29532.446,E2 -29532.446} C_VEL
LIN {X 0,Y 129.874,Z 701.222,A -85,B 0,C 180,E1 -29533.087,E2 -29533.087} C_VEL
LIN {X 0,Y 123.97,Z 712.772,A -85,B 0,C 180,E1 -29533.876,E2 -29533.876} C_VEL
LIN {X 0,Y 116.478,Z 724.417,A -85,B 0,C 180,E1 -29535.12,E2 -29535.12} C_VEL
LIN {X 0,Y 108.223,Z 734.753,A -85,B 0,C 180,E1 -29536.696,E2 -29536.696} C_VEL
LIN {X 0,Y 100.083,Z 743.139,A -85,B 0,C 180,E1 -29538.563,E2 -29538.563} C_VEL
LIN {X 0,Y 90.491,Z 751.346,A -85,B 0,C 180,E1 -29541.258,E2 -29541.258} C_VEL
LIN {X 0,Y 81.186,Z 757.967,A -85,B 0,C 180,E1 -29544.642,E2 -29544.642} C_VEL
LIN {X 0,Y 71.817,Z 763.544,A -85,B 0,C 180,E1 -29549.294,E2 -29549.294} C_VEL
LIN {X 0,Y 63.977,Z 767.391,A -85,B 0,C 180,E1 -29554.526,E2 -29554.526} C_VEL
LIN {X 0,Y 56.323,Z 770.477,A -85,B 0,C 180,E1 -29561.526,E2 -29561.526} C_VEL
LIN {X 0,Y 51.778,Z 772.021,A -85,B 0,C 180,E1 -29567.262,E2 -29567.262} C_VEL
LIN {X 0,Y 44.817,Z 773.828,A -85,B 0,C 180,E1 -29581.938,E2 -29581.938} C_VEL
LIN {X 0,Y 42.647,Z 774.155,A -85,B 0,C 180,E1 -29590.757,E2 -29590.757} C_VEL
LIN {X 0,Y 41.458,Z 774.098,A -85,B 0,C 180,E1 -29600.24,E2 -29600.24} C_VEL
LIN {X 0,Y 41.324,Z 773.617,A -85,B 0,C 180,E1 -29610,E2 -29610} C_VEL
LIN {X 0,Y 41.459,Z 772.702,A -85,B 0,C 180,E1 -29619.759,E2 -29619.759} C_VEL
LIN {X 0,Y 42.599,Z 771.388,A -85,B 0,C 180,E1 -29629.266,E2 -29629.266} C_VEL
LIN {X 0,Y 46.129,Z 768.6,A -85,B 0,C 180,E1 -29642.224,E2 -29642.224} C_VEL
LIN {X 0,Y 51.624,Z 764.786,A -85,B 0,C 180,E1 -29652.896,E2 -29652.896} C_VEL
LIN {X 0,Y 58.52,Z 759.843,A -85,B 0,C 180,E1 -29661.315,E2 -29661.315} C_VEL
LIN {X 0,Y 63.712,Z 755.872,A -85,B 0,C 180,E1 -29665.823,E2 -29665.823} C_VEL
LIN {X 0,Y 71.985,Z 748.618,A -85,B 0,C 180,E1 -29671.482,E2 -29671.482} C_VEL
LIN {X 0,Y 80.817,Z 739.61,A -85,B 0,C 180,E1 -29675.933,E2 -29675.933} C_VEL
LIN {X 0,Y 88.532,Z 730.351,A -85,B 0,C 180,E1 -29678.866,E2 -29678.866} C_VEL
LIN {X 0,Y 95.637,Z 720.033,A -85,B 0,C 180,E1 -29681.104,E2 -29681.104} C_VEL
LIN {X 0,Y 102.087,Z 708.59,A -85,B 0,C 180,E1 -29682.78,E2 -29682.78} C_VEL
LIN {X 0,Y 107.392,Z 696.662,A -85,B 0,C 180,E1 -29683.98,E2 -29683.98} C_VEL
LIN {X 0,Y 111.286,Z 684.862,A -85,B 0,C 180,E1 -29684.836,E2 -29684.836} C_VEL
LIN {X 0,Y 114.314,Z 671.43,A -85,B 0,C 180,E1 -29685.481,E2 -29685.481} C_VEL
LIN {X 0,Y 115.983,Z 658.296,A -85,B 0,C 180,E1 -29685.973,E2 -29685.973} C_VEL
LIN {X 0,Y 114.464,Z 653.89,A -85,B 0,C 180,E1 -29690.056,E2 -29690.056} C_VEL
LIN {X 0,Y 113.241,Z 650.047,A -85,B 0,C 180,E1 -29695.105,E2 -29695.105} C_VEL
LIN {X 0,Y 112.707,Z 647.321,A -85,B 0,C 180,E1 -29701.966,E2 -29701.966} C_VEL
LIN {X 0,Y 113.41,Z 650.834,A -85,B 0,C 180,E1 -29710.362,E2 -29710.362} C_VEL
LIN {X 0,Y 114.613,Z 654.371,A -85,B 0,C 180,E1 -29714.879,E2 -29714.879} C_VEL
LIN {X 0,Y 115.967,Z 658.273,A -85,B 0,C 180,E1 -29718.452,E2 -29718.452} C_VEL
LIN {X 0,Y 114.028,Z 672.222,A -85,B 0,C 180,E1 -29718.996,E2 -29718.996} C_VEL
LIN {X 0,Y 111.242,Z 683.927,A -85,B 0,C 180,E1 -29719.635,E2 -29719.635} C_VEL
LIN {X 0,Y 106.735,Z 697.064,A -85,B 0,C 180,E1 -29720.761,E2 -29720.761} C_VEL
LIN {X 0,Y 105.722,Z 699.536,A -85,B 0,C 180,E1 -29721.002,E2 -29721.002} C_VEL
LIN {X 0,Y 103.94,Z 703.122,A -85,B 0,C 180,E1 -29721.024,E2 -29721.024} C_VEL
LIN {X 0,Y 96.505,Z 714.045,A -85,B 0,C 180,E1 -29719.343,E2 -29719.343} C_VEL
LIN {X 0,Y 94.308,Z 717.329,A -85,B 0,C 180,E1 -29719.509,E2 -29719.509} C_VEL
LIN {X 0,Y 86.981,Z 727.9,A -85,B 0,C 180,E1 -29721.694,E2 -29721.694} C_VEL
LIN {X 0,Y 79.016,Z 737.214,A -85,B 0,C 180,E1 -29724.264,E2 -29724.264} C_VEL
LIN {X 0,Y 69.77,Z 746.201,A -85,B 0,C 180,E1 -29728.192,E2 -29728.192} C_VEL
LIN {X 0,Y 61.062,Z 753.431,A -85,B 0,C 180,E1 -29733.444,E2 -29733.444} C_VEL
LIN {X 0,Y 51.606,Z 760.056,A -85,B 0,C 180,E1 -29741.496,E2 -29741.496} C_VEL
LIN {X 0,Y 44.512,Z 764.435,A -85,B 0,C 180,E1 -29750.835,E2 -29750.835} C_VEL
LIN {X 0,Y 40.491,Z 766.754,A -85,B 0,C 180,E1 -29758.621,E2 -29758.621} C_VEL
LIN {X 0,Y 37.357,Z 768.646,A -85,B 0,C 180,E1 -29767.898,E2 -29767.898} C_VEL
LIN {X 0,Y 35.228,Z 770.105,A -85,B 0,C 180,E1 -29778.493,E2 -29778.493} C_VEL
LIN {X 0,Y 34.243,Z 771.135,A -85,B 0,C 180,E1 -29790,E2 -29790} C_VEL
LIN {X 0,Y 34.399,Z 771.789,A -85,B 0,C 180,E1 -29801.789,E2 -29801.789} C_VEL
LIN {X 0,Y 35.795,Z 772.065,A -85,B 0,C 180,E1 -29813.121,E2 -29813.121} C_VEL
LIN {X 0,Y 38.336,Z 771.937,A -85,B 0,C 180,E1 -29823.365,E2 -29823.365} C_VEL
LIN {X 0,Y 46.25,Z 770.45,A -85,B 0,C 180,E1 -29839.444,E2 -29839.444} C_VEL
LIN {X 0,Y 55.358,Z 767.767,A -85,B 0,C 180,E1 -29849.48,E2 -29849.48} C_VEL
LIN {X 0,Y 65.233,Z 763.848,A -85,B 0,C 180,E1 -29856.312,E2 -29856.312} C_VEL
LIN {X 0,Y 74.409,Z 759.231,A -85,B 0,C 180,E1 -29860.82,E2 -29860.82} C_VEL
LIN {X 0,Y 85.592,Z 752.241,A -85,B 0,C 180,E1 -29864.747,E2 -29864.747} C_VEL
LIN {X 0,Y 95.359,Z 744.658,A -85,B 0,C 180,E1 -29867.557,E2 -29867.557} C_VEL
LIN {X 0,Y 103.665,Z 736.876,A -85,B 0,C 180,E1 -29869.422,E2 -29869.422} C_VEL
LIN {X 0,Y 112.077,Z 727.352,A -85,B 0,C 180,E1 -29870.97,E2 -29870.97} C_VEL
LIN {X 0,Y 119.704,Z 716.764,A -85,B 0,C 180,E1 -29872.193,E2 -29872.193} C_VEL
LIN {X 0,Y 126.509,Z 704.893,A -85,B 0,C 180,E1 -29873.211,E2 -29873.211} C_VEL
LIN {X 0,Y 131.836,Z 692.708,A -85,B 0,C 180,E1 -29873.98,E2 -29873.98} C_VEL
LIN {X 0,Y 135.206,Z 682.538,A -85,B 0,C 180,E1 -29874.453,E2 -29874.453} C_VEL
LIN {X 0,Y 135.092,Z 680.565,A -85,B 0,C 180,E1 -29877.391,E2 -29877.391} C_VEL
LIN {X 0,Y 135.098,Z 679.453,A -85,B 0,C 180,E1 -29880,E2 -29880} C_VEL
LIN {X 0,Y 135.099,Z 679.497,A -85,B 0,C 180,E1 -29883.355,E2 -29883.355} C_VEL
LIN {X 0,Y 135.228,Z 681.694,A -85,B 0,C 180,E1 -29887.841,E2 -29887.841} C_VEL
LIN {X 0,Y 135.266,Z 682.911,A -85,B 0,C 180,E1 -29889.193,E2 -29889.193} C_VEL
LIN {X 0,Y 130.834,Z 695.998,A -85,B 0,C 180,E1 -29889.707,E2 -29889.707} C_VEL
LIN {X 0,Y 125.88,Z 706.812,A -85,B 0,C 180,E1 -29890.263,E2 -29890.263} C_VEL
LIN {X 0,Y 119.065,Z 718.445,A -85,B 0,C 180,E1 -29891.1,E2 -29891.1} C_VEL
LIN {X 0,Y 111.451,Z 728.911,A -85,B 0,C 180,E1 -29892.207,E2 -29892.207} C_VEL
LIN {X 0,Y 103.054,Z 738.349,A -85,B 0,C 180,E1 -29893.643,E2 -29893.643} C_VEL
LIN {X 0,Y 93.087,Z 747.447,A -85,B 0,C 180,E1 -29895.722,E2 -29895.722} C_VEL
LIN {X 0,Y 83.294,Z 754.789,A -85,B 0,C 180,E1 -29898.341,E2 -29898.341} C_VEL
LIN {X 0,Y 72.202,Z 761.547,A -85,B 0,C 180,E1 -29902.379,E2 -29902.379} C_VEL
LIN {X 0,Y 63.157,Z 766.024,A -85,B 0,C 180,E1 -29907.102,E2 -29907.102} C_VEL
LIN {X 0,Y 57.339,Z 768.39,A -85,B 0,C 180,E1 -29910.911,E2 -29910.911} C_VEL
LIN {X 0,Y 51.872,Z 770.334,A -85,B 0,C 180,E1 -29915.619,E2 -29915.619} C_VEL
LIN {X 0,Y 46.806,Z 771.861,A -85,B 0,C 180,E1 -29921.345,E2 -29921.345} C_VEL
LIN {X 0,Y 38.672,Z 773.64,A -85,B 0,C 180,E1 -29936.962,E2 -29936.962} C_VEL
LIN {X 0,Y 36.003,Z 773.955,A -85,B 0,C 180,E1 -29947.02,E2 -29947.02} C_VEL
LIN {X 0,Y 34.481,Z 773.885,A -85,B 0,C 180,E1 -29958.24,E2 -29958.24} C_VEL
LIN {X 0,Y 34.239,Z 773.385,A -85,B 0,C 180,E1 -29970,E2 -29970} C_VEL
LIN {X 0,Y 34.477,Z 772.458,A -85,B 0,C 180,E1 -29981.762,E2 -29981.762} C_VEL
LIN {X 0,Y 35.957,Z 771.132,A -85,B 0,C 180,E1 -29993.011,E2 -29993.011} C_VEL
LIN {X 0,Y 40.267,Z 768.319,A -85,B 0,C 180,E1 -30007.651,E2 -30007.651} C_VEL
LIN {X 0,Y 46.649,Z 764.479,A -85,B 0,C 180,E1 -30018.874,E2 -30018.874} C_VEL
LIN {X 0,Y 54.357,Z 759.51,A -85,B 0,C 180,E1 -30027.18,E2 -30027.18} C_VEL
LIN {X 0,Y 62.859,Z 753.254,A -85,B 0,C 180,E1 -30033.435,E2 -30033.435} C_VEL
LIN {X 0,Y 71.906,Z 745.434,A -85,B 0,C 180,E1 -30038.201,E2 -30038.201} C_VEL
LIN {X 0,Y 81.365,Z 735.652,A -85,B 0,C 180,E1 -30041.825,E2 -30041.825} C_VEL
LIN {X 0,Y 89.47,Z 725.522,A -85,B 0,C 180,E1 -30044.202,E2 -30044.202} C_VEL
LIN {X 0,Y 96.885,Z 714.037,A -85,B 0,C 180,E1 -30045.976,E2 -30045.976} C_VEL
LIN {X 0,Y 102.716,Z 702.755,A -85,B 0,C 180,E1 -30047.159,E2 -30047.159} C_VEL
LIN {X 0,Y 107.301,Z 691.274,A -85,B 0,C 180,E1 -30048.057,E2 -30048.057} C_VEL
LIN {X 0,Y 111.135,Z 677.894,A -85,B 0,C 180,E1 -30048.719,E2 -30048.719} C_VEL
LIN {X 0,Y 113.443,Z 665.008,A -85,B 0,C 180,E1 -30049.143,E2 -30049.143} C_VEL
LIN {X 0,Y 113.722,Z 662.385,A -85,B 0,C 180,E1 -30049.316,E2 -30049.316} C_VEL
LIN {X 0,Y 112.709,Z 658.966,A -85,B 0,C 180,E1 -30053.061,E2 -30053.061} C_VEL
LIN {X 0,Y 112.128,Z 656.703,A -85,B 0,C 180,E1 -30056.407,E2 -30056.407} C_VEL
LIN {X 0,Y 111.804,Z 654.743,A -85,B 0,C 180,E1 -30061.486,E2 -30061.486} C_VEL
LIN {X 0,Y 111.779,Z 655.037,A -85,B 0,C 180,E1 -30063.34,E2 -30063.34} C_VEL
LIN {X 0,Y 112.321,Z 657.678,A -85,B 0,C 180,E1 -30069.454,E2 -30069.454} C_VEL
LIN {X 0,Y 113.156,Z 660.551,A -85,B 0,C 180,E1 -30073.24,E2 -30073.24} C_VEL
LIN {X 0,Y 113.718,Z 662.358,A -85,B 0,C 180,E1 -30075.128,E2 -30075.128} C_VEL
LIN {X 0,Y 111.58,Z 675.167,A -85,B 0,C 180,E1 -30075.632,E2 -30075.632} C_VEL
LIN {X 0,Y 108.188,Z 687.727,A -85,B 0,C 180,E1 -30076.348,E2 -30076.348} C_VEL
LIN {X 0,Y 103.588,Z 699.853,A -85,B 0,C 180,E1 -30077.301,E2 -30077.301} C_VEL
LIN {X 0,Y 98.188,Z 710.759,A -85,B 0,C 180,E1 -30078.492,E2 -30078.492} C_VEL
LIN {X 0,Y 94.308,Z 717.329,A -85,B 0,C 180,E1 -30079.509,E2 -30079.509} C_VEL
LIN {X 0,Y 90.969,Z 722.169,A -85,B 0,C 180,E1 -30080.034,E2 -30080.034} C_VEL
LIN {X 0,Y 84.494,Z 729.703,A -85,B 0,C 180,E1 -30079.883,E2 -30079.883} C_VEL
LIN {X 0,Y 77.464,Z 736.764,A -85,B 0,C 180,E1 -30079.719,E2 -30079.719} C_VEL
LIN {X 0,Y 73.258,Z 740.751,A -85,B 0,C 180,E1 -30080.398,E2 -30080.398} C_VEL
LIN {X 0,Y 65.155,Z 747.937,A -85,B 0,C 180,E1 -30083.532,E2 -30083.532} C_VEL
LIN {X 0,Y 55.953,Z 754.842,A -85,B 0,C 180,E1 -30088.452,E2 -30088.452} C_VEL
LIN {X 0,Y 47.213,Z 760.376,A -85,B 0,C 180,E1 -30095.046,E2 -30095.046} C_VEL
LIN {X 0,Y 39.268,Z 764.729,A -85,B 0,C 180,E1 -30104.284,E2 -30104.284} C_VEL
LIN {X 0,Y 34.64,Z 767.035,A -85,B 0,C 180,E1 -30112.509,E2 -30112.509} C_VEL
LIN {X 0,Y 30.919,Z 768.914,A -85,B 0,C 180,E1 -30122.961,E2 -30122.961} C_VEL
LIN {X 0,Y 28.306,Z 770.35,A -85,B 0,C 180,E1 -30135.624,E2 -30135.624} C_VEL
LIN {X 0,Y 27.123,Z 771.37,A -85,B 0,C 180,E1 -30150,E2 -30150} C_VEL
LIN {X 0,Y 27.469,Z 772.012,A -85,B 0,C 180,E1 -30164.824,E2 -30164.824} C_VEL
LIN {X 0,Y 29.366,Z 772.276,A -85,B 0,C 180,E1 -30178.597,E2 -30178.597} C_VEL
LIN {X 0,Y 32.59,Z 772.127,A -85,B 0,C 180,E1 -30190.31,E2 -30190.31} C_VEL
LIN {X 0,Y 41.949,Z 770.616,A -85,B 0,C 180,E1 -30206.894,E2 -30206.894} C_VEL
LIN {X 0,Y 51.301,Z 768.141,A -85,B 0,C 180,E1 -30215.732,E2 -30215.732} C_VEL
LIN {X 0,Y 62.696,Z 763.951,A -85,B 0,C 180,E1 -30222.324,E2 -30222.324} C_VEL
LIN {X 0,Y 72.374,Z 759.306,A -85,B 0,C 180,E1 -30226.177,E2 -30226.177} C_VEL
LIN {X 0,Y 82.323,Z 753.4,A -85,B 0,C 180,E1 -30229.036,E2 -30229.036} C_VEL
LIN {X 0,Y 92.382,Z 746.025,A -85,B 0,C 180,E1 -30231.476,E2 -30231.476} C_VEL
LIN {X 0,Y 100.887,Z 738.492,A -85,B 0,C 180,E1 -30233.056,E2 -30233.056} C_VEL
LIN {X 0,Y 109.457,Z 729.355,A -85,B 0,C 180,E1 -30234.383,E2 -30234.383} C_VEL
LIN {X 0,Y 117.218,Z 719.187,A -85,B 0,C 180,E1 -30235.381,E2 -30235.381} C_VEL
LIN {X 0,Y 124.135,Z 707.871,A -85,B 0,C 180,E1 -30236.224,E2 -30236.224} C_VEL
LIN {X 0,Y 129.67,Z 696.334,A -85,B 0,C 180,E1 -30236.893,E2 -30236.893} C_VEL
LIN {X 0,Y 132.968,Z 687.466,A -85,B 0,C 180,E1 -30237.348,E2 -30237.348} C_VEL
LIN {X 0,Y 133.029,Z 686.39,A -85,B 0,C 180,E1 -30240,E2 -30240} C_VEL
LIN {X 0,Y 133.079,Z 686.262,A -85,B 0,C 180,E1 -30243.027,E2 -30243.027} C_VEL
LIN {X 0,Y 133.016,Z 687.578,A -85,B 0,C 180,E1 -30246.066,E2 -30246.066} C_VEL
LIN {X 0,Y 132.657,Z 688.805,A -85,B 0,C 180,E1 -30246.358,E2 -30246.358} C_VEL
LIN {X 0,Y 127.932,Z 700.748,A -85,B 0,C 180,E1 -30246.822,E2 -30246.822} C_VEL
LIN {X 0,Y 122.213,Z 711.743,A -85,B 0,C 180,E1 -30247.273,E2 -30247.273} C_VEL
LIN {X 0,Y 114.471,Z 723.496,A -85,B 0,C 180,E1 -30248.118,E2 -30248.118} C_VEL
LIN {X 0,Y 106.742,Z 732.975,A -85,B 0,C 180,E1 -30249.036,E2 -30249.036} C_VEL
LIN {X 0,Y 98.202,Z 741.635,A -85,B 0,C 180,E1 -30250.257,E2 -30250.257} C_VEL
LIN {X 0,Y 88.047,Z 750.051,A -85,B 0,C 180,E1 -30252.1,E2 -30252.1} C_VEL
LIN {X 0,Y 78.021,Z 756.832,A -85,B 0,C 180,E1 -30254.461,E2 -30254.461} C_VEL
LIN {X 0,Y 66.574,Z 763.077,A -85,B 0,C 180,E1 -30258.182,E2 -30258.182} C_VEL
LIN {X 0,Y 57.131,Z 767.156,A -85,B 0,C 180,E1 -30262.693,E2 -30262.693} C_VEL
LIN {X 0,Y 48.066,Z 770.192,A -85,B 0,C 180,E1 -30268.684,E2 -30268.684} C_VEL
LIN {X 0,Y 42.447,Z 771.699,A -85,B 0,C 180,E1 -30274.124,E2 -30274.124} C_VEL
LIN {X 0,Y 32.931,Z 773.451,A -85,B 0,C 180,E1 -30290.19,E2 -30290.19} C_VEL
LIN {X 0,Y 29.588,Z 773.756,A -85,B 0,C 180,E1 -30301.637,E2 -30301.637} C_VEL
LIN {X 0,Y 27.55,Z 773.669,A -85,B 0,C 180,E1 -30315.221,E2 -30315.221} C_VEL
LIN {X 0,Y 27.125,Z 773.151,A -85,B 0,C 180,E1 -30330,E2 -30330} C_VEL
LIN {X 0,Y 27.544,Z 772.212,A -85,B 0,C 180,E1 -30344.783,E2 -30344.783} C_VEL
LIN {X 0,Y 29.518,Z 770.874,A -85,B 0,C 180,E1 -30358.436,E2 -30358.436} C_VEL
LIN {X 0,Y 34.893,Z 768.038,A -85,B 0,C 180,E1 -30374.825,E2 -30374.825} C_VEL
LIN {X 0,Y 42.302,Z 764.173,A -85,B 0,C 180,E1 -30386.169,E2 -30386.169} C_VEL
LIN {X 0,Y 50.855,Z 759.177,A -85,B 0,C 180,E1 -30393.929,E2 -30393.929} C_VEL
LIN {X 0,Y 60.007,Z 752.89,A -85,B 0,C 180,E1 -30399.542,E2 -30399.542} C_VEL
LIN {X 0,Y 69.568,Z 745.016,A -85,B 0,C 180,E1 -30403.678,E2 -30403.678} C_VEL
LIN {X 0,Y 79.432,Z 735.194,A -85,B 0,C 180,E1 -30406.713,E2 -30406.713} C_VEL
LIN {X 0,Y 87.803,Z 724.987,A -85,B 0,C 180,E1 -30408.665,E2 -30408.665} C_VEL
LIN {X 0,Y 95.41,Z 713.428,A -85,B 0,C 180,E1 -30410.127,E2 -30410.127} C_VEL
LIN {X 0,Y 101.368,Z 702.063,A -85,B 0,C 180,E1 -30411.076,E2 -30411.076} C_VEL
LIN {X 0,Y 106.07,Z 690.337,A -85,B 0,C 180,E1 -30411.812,E2 -30411.812} C_VEL
LIN {X 0,Y 109.854,Z 677.137,A -85,B 0,C 180,E1 -30412.335,E2 -30412.335} C_VEL
LIN {X 0,Y 111.781,Z 666.869,A -85,B 0,C 180,E1 -30412.652,E2 -30412.652} C_VEL
LIN {X 0,Y 111.124,Z 663.509,A -85,B 0,C 180,E1 -30417.282,E2 -30417.282} C_VEL
LIN {X 0,Y 110.919,Z 662.541,A -85,B 0,C 180,E1 -30420,E2 -30420} C_VEL
LIN {X 0,Y 110.891,Z 662.569,A -85,B 0,C 180,E1 -30424.089,E2 -30424.089} C_VEL
LIN {X 0,Y 111.242,Z 664.519,A -85,B 0,C 180,E1 -30428.63,E2 -30428.63} C_VEL
LIN {X 0,Y 111.729,Z 666.814,A -85,B 0,C 180,E1 -30431.7,E2 -30431.7} C_VEL
LIN {X 0,Y 109.138,Z 679.529,A -85,B 0,C 180,E1 -30432.187,E2 -30432.187} C_VEL
LIN {X 0,Y 104.928,Z 692.826,A -85,B 0,C 180,E1 -30432.972,E2 -30432.972} C_VEL
